REGION Network 3: Avoidance
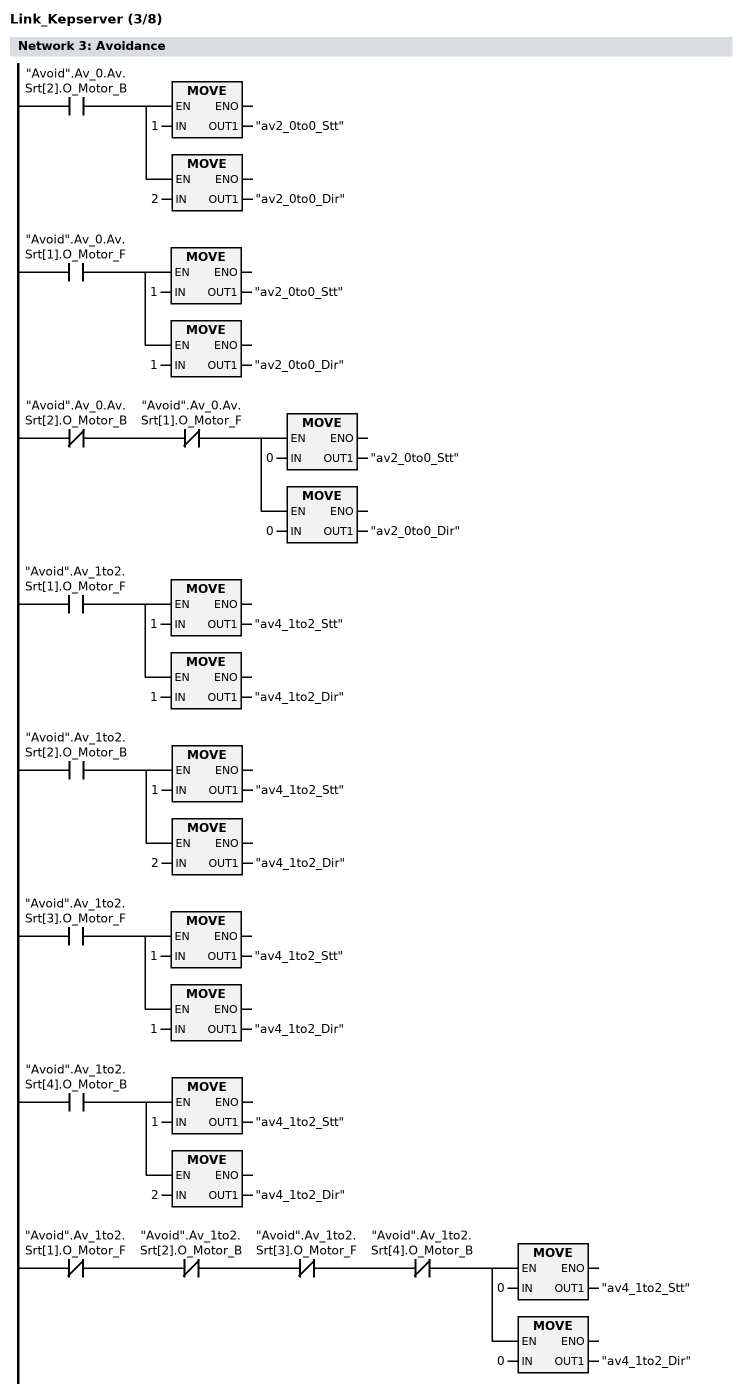
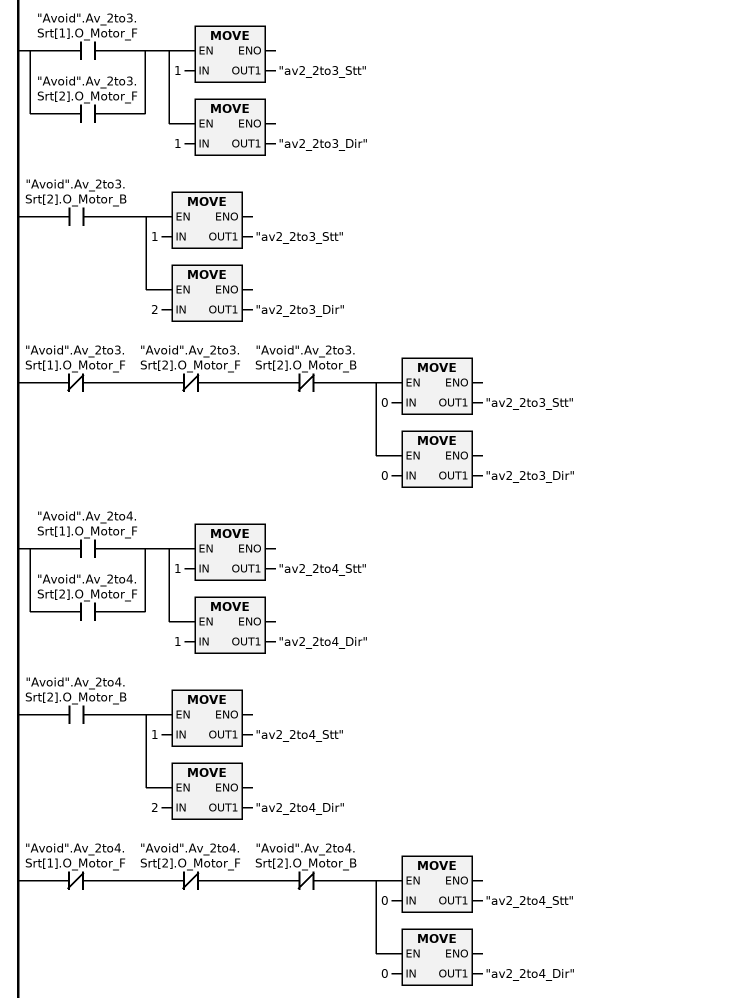
   RUNG wire#powerrail
      Contact( "Avoid".Av_0.Av.Srt[2].O_Motor_B )
      wire#w1
      Move(in := 1, out1 => "av2_0to0_Stt")
   END_RUNG
   RUNG wire#w1
      Move(in := 2, out1 => "av2_0to0_Dir")
   END_RUNG
   RUNG wire#powerrail
      Contact( "Avoid".Av_0.Av.Srt[1].O_Motor_F )
      wire#w2
      Move(in := 1, out1 => "av2_0to0_Stt")
   END_RUNG
   RUNG wire#w2
      Move(in := 1, out1 => "av2_0to0_Dir")
   END_RUNG
   RUNG wire#powerrail
      I_Contact( "Avoid".Av_0.Av.Srt[2].O_Motor_B )
      I_Contact( "Avoid".Av_0.Av.Srt[1].O_Motor_F )
      wire#w3
      Move(in := 0, out1 => "av2_0to0_Stt")
   END_RUNG
   RUNG wire#w3
      Move(in := 0, out1 => "av2_0to0_Dir")
   END_RUNG
   RUNG wire#powerrail
      Contact( "Avoid".Av_1to2.Srt[1].O_Motor_F )
      wire#w4
      Move(in := 1, out1 => "av4_1to2_Stt")
   END_RUNG
   RUNG wire#w4
      Move(in := 1, out1 => "av4_1to2_Dir")
   END_RUNG
   RUNG wire#powerrail
      Contact( "Avoid".Av_1to2.Srt[2].O_Motor_B )
      wire#w5
      Move(in := 1, out1 => "av4_1to2_Stt")
   END_RUNG
   RUNG wire#w5
      Move(in := 2, out1 => "av4_1to2_Dir")
   END_RUNG
   RUNG wire#powerrail
      Contact( "Avoid".Av_1to2.Srt[3].O_Motor_F )
      wire#w6
      Move(in := 1, out1 => "av4_1to2_Stt")
   END_RUNG
   RUNG wire#w6
      Move(in := 1, out1 => "av4_1to2_Dir")
   END_RUNG
   RUNG wire#powerrail
      Contact( "Avoid".Av_1to2.Srt[4].O_Motor_B )
      wire#w7
      Move(in := 1, out1 => "av4_1to2_Stt")
   END_RUNG
   RUNG wire#w7
      Move(in := 2, out1 => "av4_1to2_Dir")
   END_RUNG
   RUNG wire#powerrail
      I_Contact( "Avoid".Av_1to2.Srt[1].O_Motor_F )
      I_Contact( "Avoid".Av_1to2.Srt[2].O_Motor_B )
      I_Contact( "Avoid".Av_1to2.Srt[3].O_Motor_F )
      I_Contact( "Avoid".Av_1to2.Srt[4].O_Motor_B )
      wire#w8
      Move(in := 0, out1 => "av4_1to2_Stt")
   END_RUNG
   RUNG wire#w8
      Move(in := 0, out1 => "av4_1to2_Dir")
   END_RUNG
   RUNG wire#powerrail
      Contact( "Avoid".Av_2to3.Srt[1].O_Motor_F )
      wire#w9
      Move(in := 1, out1 => "av2_2to3_Stt")
   END_RUNG
   RUNG wire#powerrail
      Contact( "Avoid".Av_2to3.Srt[2].O_Motor_F )
   END_RUNG wire#w9
   RUNG wire#w9
      Move(in := 1, out1 => "av2_2to3_Dir")
   END_RUNG
   RUNG wire#powerrail
      Contact( "Avoid".Av_2to3.Srt[2].O_Motor_B )
      wire#w10
      Move(in := 1, out1 => "av2_2to3_Stt")
   END_RUNG
   RUNG wire#w10
      Move(in := 2, out1 => "av2_2to3_Dir")
   END_RUNG
   RUNG wire#powerrail
      I_Contact( "Avoid".Av_2to3.Srt[1].O_Motor_F )
      I_Contact( "Avoid".Av_2to3.Srt[2].O_Motor_F )
      I_Contact( "Avoid".Av_2to3.Srt[2].O_Motor_B )
      wire#w11
      Move(in := 0, out1 => "av2_2to3_Stt")
   END_RUNG
   RUNG wire#w11
      Move(in := 0, out1 => "av2_2to3_Dir")
   END_RUNG
   RUNG wire#powerrail
      Contact( "Avoid".Av_2to4.Srt[1].O_Motor_F )
      wire#w12
      Move(in := 1, out1 => "av2_2to4_Stt")
   END_RUNG
   RUNG wire#powerrail
      Contact( "Avoid".Av_2to4.Srt[2].O_Motor_F )
   END_RUNG wire#w12
   RUNG wire#w12
      Move(in := 1, out1 => "av2_2to4_Dir")
   END_RUNG
   RUNG wire#powerrail
      Contact( "Avoid".Av_2to4.Srt[2].O_Motor_B )
      wire#w13
      Move(in := 1, out1 => "av2_2to4_Stt")
   END_RUNG
   RUNG wire#w13
      Move(in := 2, out1 => "av2_2to4_Dir")
   END_RUNG
   RUNG wire#powerrail
      I_Contact( "Avoid".Av_2to4.Srt[1].O_Motor_F )
      I_Contact( "Avoid".Av_2to4.Srt[2].O_Motor_F )
      I_Contact( "Avoid".Av_2to4.Srt[2].O_Motor_B )
      wire#w14
      Move(in := 0, out1 => "av2_2to4_Stt")
   END_RUNG
   RUNG wire#w14
      Move(in := 0, out1 => "av2_2to4_Dir")
   END_RUNG
   // the same network as SCL:
   IF "Avoid".Av_0.Av.Srt[2].O_Motor_B THEN
       "av2_0to0_Stt" := 1;
       "av2_0to0_Dir" := 2;
   END_IF;
   IF "Avoid".Av_0.Av.Srt[1].O_Motor_F THEN
       "av2_0to0_Stt" := 1;
       "av2_0to0_Dir" := 1;
   END_IF;
   IF NOT "Avoid".Av_0.Av.Srt[2].O_Motor_B AND NOT "Avoid".Av_0.Av.Srt[1].O_Motor_F THEN
       "av2_0to0_Stt" := 0;
       "av2_0to0_Dir" := 0;
   END_IF;
   IF "Avoid".Av_1to2.Srt[1].O_Motor_F THEN
       "av4_1to2_Stt" := 1;
       "av4_1to2_Dir" := 1;
   END_IF;
   IF "Avoid".Av_1to2.Srt[2].O_Motor_B THEN
       "av4_1to2_Stt" := 1;
       "av4_1to2_Dir" := 2;
   END_IF;
   IF "Avoid".Av_1to2.Srt[3].O_Motor_F THEN
       "av4_1to2_Stt" := 1;
       "av4_1to2_Dir" := 1;
   END_IF;
   IF "Avoid".Av_1to2.Srt[4].O_Motor_B THEN
       "av4_1to2_Stt" := 1;
       "av4_1to2_Dir" := 2;
   END_IF;
   IF NOT "Avoid".Av_1to2.Srt[1].O_Motor_F AND NOT "Avoid".Av_1to2.Srt[2].O_Motor_B AND NOT "Avoid".Av_1to2.Srt[3].O_Motor_F AND NOT "Avoid".Av_1to2.Srt[4].O_Motor_B THEN
       "av4_1to2_Stt" := 0;
       "av4_1to2_Dir" := 0;
   END_IF;
   IF "Avoid".Av_2to3.Srt[1].O_Motor_F OR "Avoid".Av_2to3.Srt[2].O_Motor_F THEN
       "av2_2to3_Stt" := 1;
       "av2_2to3_Dir" := 1;
   END_IF;
   IF "Avoid".Av_2to3.Srt[2].O_Motor_B THEN
       "av2_2to3_Stt" := 1;
       "av2_2to3_Dir" := 2;
   END_IF;
   IF NOT "Avoid".Av_2to3.Srt[1].O_Motor_F AND NOT "Avoid".Av_2to3.Srt[2].O_Motor_F AND NOT "Avoid".Av_2to3.Srt[2].O_Motor_B THEN
       "av2_2to3_Stt" := 0;
       "av2_2to3_Dir" := 0;
   END_IF;
   IF "Avoid".Av_2to4.Srt[1].O_Motor_F OR "Avoid".Av_2to4.Srt[2].O_Motor_F THEN
       "av2_2to4_Stt" := 1;
       "av2_2to4_Dir" := 1;
   END_IF;
   IF "Avoid".Av_2to4.Srt[2].O_Motor_B THEN
       "av2_2to4_Stt" := 1;
       "av2_2to4_Dir" := 2;
   END_IF;
   IF NOT "Avoid".Av_2to4.Srt[1].O_Motor_F AND NOT "Avoid".Av_2to4.Srt[2].O_Motor_F AND NOT "Avoid".Av_2to4.Srt[2].O_Motor_B THEN
       "av2_2to4_Stt" := 0;
       "av2_2to4_Dir" := 0;
   END_IF;
END_REGION

REGION Network 4: Updown
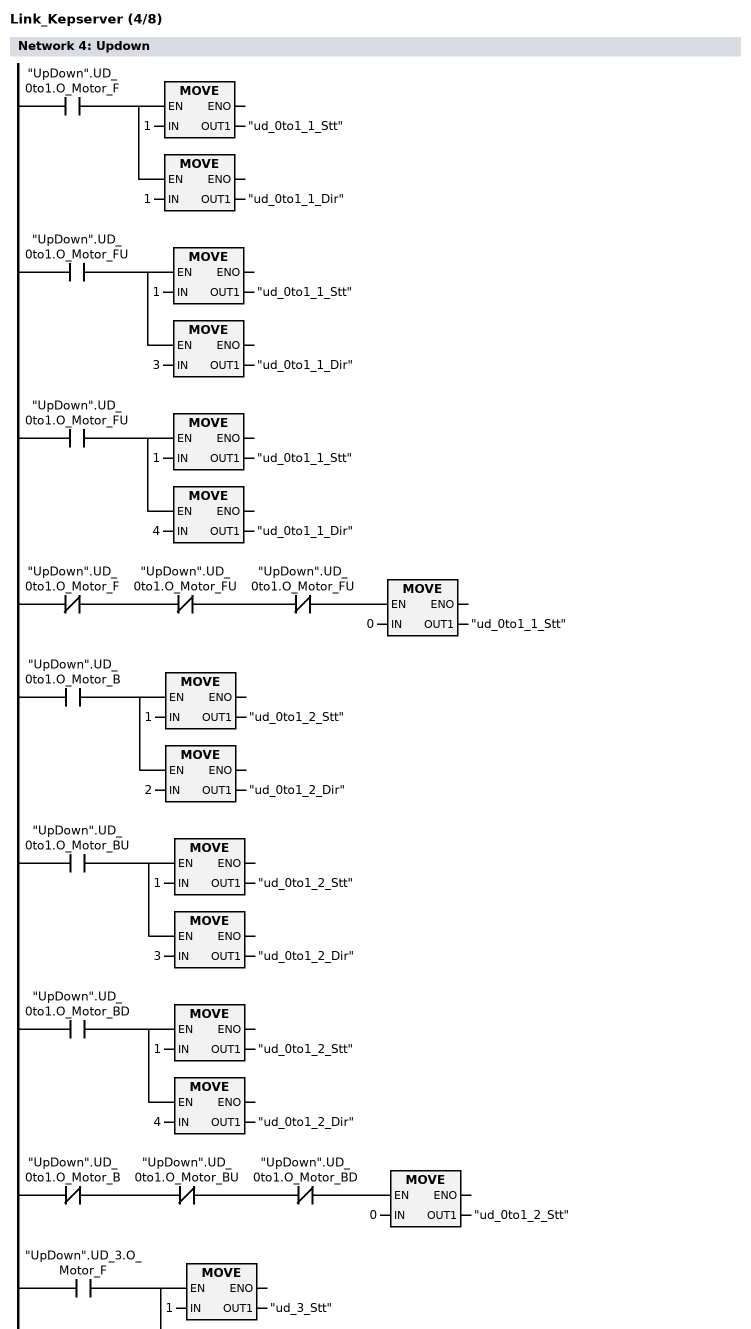
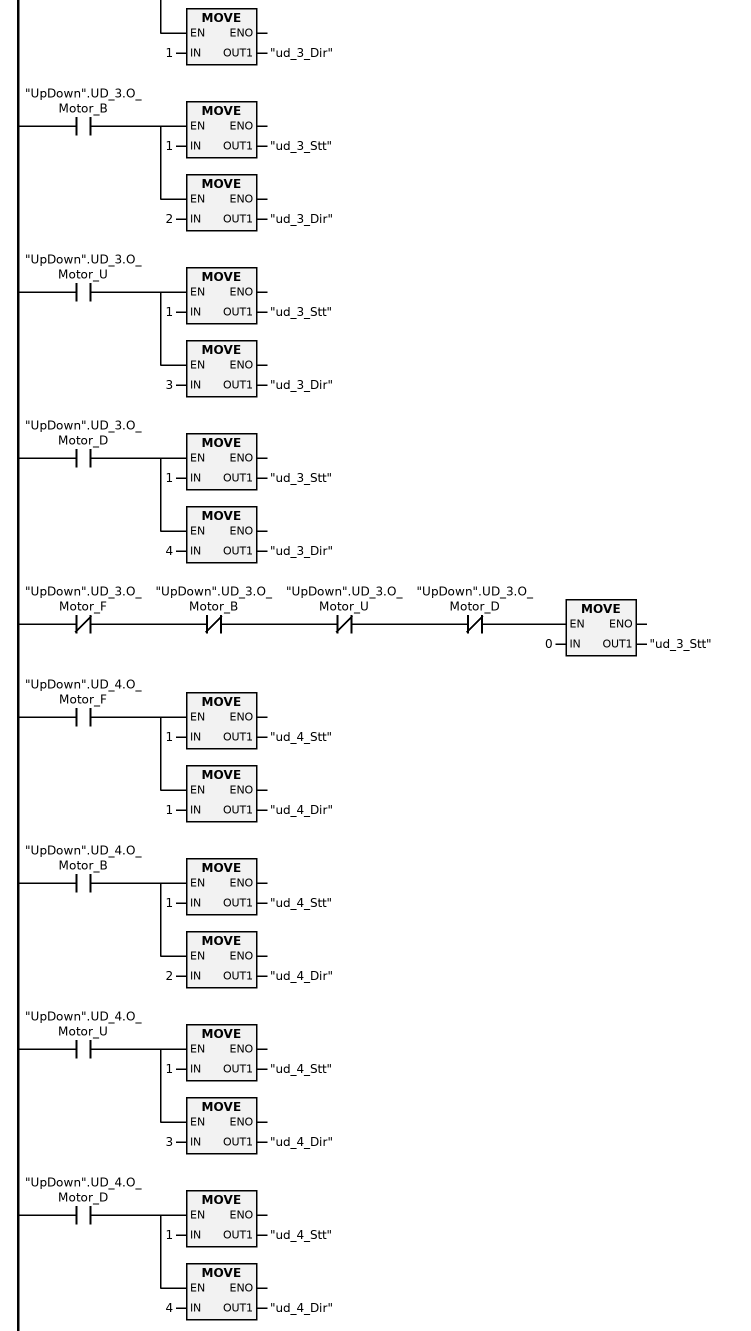
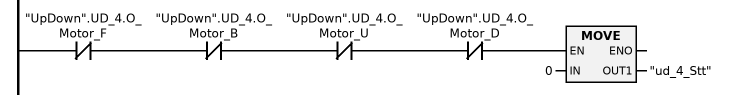
   RUNG wire#powerrail
      Contact( "UpDown".UD_0to1.O_Motor_F )
      wire#w1
      Move(in := 1, out1 => "ud_0to1_1_Stt")
   END_RUNG
   RUNG wire#w1
      Move(in := 1, out1 => "ud_0to1_1_Dir")
   END_RUNG
   RUNG wire#powerrail
      Contact( "UpDown".UD_0to1.O_Motor_FU )
      wire#w2
      Move(in := 1, out1 => "ud_0to1_1_Stt")
   END_RUNG
   RUNG wire#w2
      Move(in := 3, out1 => "ud_0to1_1_Dir")
   END_RUNG
   RUNG wire#powerrail
      Contact( "UpDown".UD_0to1.O_Motor_FU )
      wire#w3
      Move(in := 1, out1 => "ud_0to1_1_Stt")
   END_RUNG
   RUNG wire#w3
      Move(in := 4, out1 => "ud_0to1_1_Dir")
   END_RUNG
   RUNG wire#powerrail
      I_Contact( "UpDown".UD_0to1.O_Motor_F )
      I_Contact( "UpDown".UD_0to1.O_Motor_FU )
      I_Contact( "UpDown".UD_0to1.O_Motor_FU )
      Move(in := 0, out1 => "ud_0to1_1_Stt")
   END_RUNG
   RUNG wire#powerrail
      Contact( "UpDown".UD_0to1.O_Motor_B )
      wire#w4
      Move(in := 1, out1 => "ud_0to1_2_Stt")
   END_RUNG
   RUNG wire#w4
      Move(in := 2, out1 => "ud_0to1_2_Dir")
   END_RUNG
   RUNG wire#powerrail
      Contact( "UpDown".UD_0to1.O_Motor_BU )
      wire#w5
      Move(in := 1, out1 => "ud_0to1_2_Stt")
   END_RUNG
   RUNG wire#w5
      Move(in := 3, out1 => "ud_0to1_2_Dir")
   END_RUNG
   RUNG wire#powerrail
      Contact( "UpDown".UD_0to1.O_Motor_BD )
      wire#w6
      Move(in := 1, out1 => "ud_0to1_2_Stt")
   END_RUNG
   RUNG wire#w6
      Move(in := 4, out1 => "ud_0to1_2_Dir")
   END_RUNG
   RUNG wire#powerrail
      I_Contact( "UpDown".UD_0to1.O_Motor_B )
      I_Contact( "UpDown".UD_0to1.O_Motor_BU )
      I_Contact( "UpDown".UD_0to1.O_Motor_BD )
      Move(in := 0, out1 => "ud_0to1_2_Stt")
   END_RUNG
   RUNG wire#powerrail
      Contact( "UpDown".UD_3.O_Motor_F )
      wire#w7
      Move(in := 1, out1 => "ud_3_Stt")
   END_RUNG
   RUNG wire#w7
      Move(in := 1, out1 => "ud_3_Dir")
   END_RUNG
   RUNG wire#powerrail
      Contact( "UpDown".UD_3.O_Motor_B )
      wire#w8
      Move(in := 1, out1 => "ud_3_Stt")
   END_RUNG
   RUNG wire#w8
      Move(in := 2, out1 => "ud_3_Dir")
   END_RUNG
   RUNG wire#powerrail
      Contact( "UpDown".UD_3.O_Motor_U )
      wire#w9
      Move(in := 1, out1 => "ud_3_Stt")
   END_RUNG
   RUNG wire#w9
      Move(in := 3, out1 => "ud_3_Dir")
   END_RUNG
   RUNG wire#powerrail
      Contact( "UpDown".UD_3.O_Motor_D )
      wire#w10
      Move(in := 1, out1 => "ud_3_Stt")
   END_RUNG
   RUNG wire#w10
      Move(in := 4, out1 => "ud_3_Dir")
   END_RUNG
   RUNG wire#powerrail
      I_Contact( "UpDown".UD_3.O_Motor_F )
      I_Contact( "UpDown".UD_3.O_Motor_B )
      I_Contact( "UpDown".UD_3.O_Motor_U )
      I_Contact( "UpDown".UD_3.O_Motor_D )
      Move(in := 0, out1 => "ud_3_Stt")
   END_RUNG
   RUNG wire#powerrail
      Contact( "UpDown".UD_4.O_Motor_F )
      wire#w11
      Move(in := 1, out1 => "ud_4_Stt")
   END_RUNG
   RUNG wire#w11
      Move(in := 1, out1 => "ud_4_Dir")
   END_RUNG
   RUNG wire#powerrail
      Contact( "UpDown".UD_4.O_Motor_B )
      wire#w12
      Move(in := 1, out1 => "ud_4_Stt")
   END_RUNG
   RUNG wire#w12
      Move(in := 2, out1 => "ud_4_Dir")
   END_RUNG
   RUNG wire#powerrail
      Contact( "UpDown".UD_4.O_Motor_U )
      wire#w13
      Move(in := 1, out1 => "ud_4_Stt")
   END_RUNG
   RUNG wire#w13
      Move(in := 3, out1 => "ud_4_Dir")
   END_RUNG
   RUNG wire#powerrail
      Contact( "UpDown".UD_4.O_Motor_D )
      wire#w14
      Move(in := 1, out1 => "ud_4_Stt")
   END_RUNG
   RUNG wire#w14
      Move(in := 4, out1 => "ud_4_Dir")
   END_RUNG
   RUNG wire#powerrail
      I_Contact( "UpDown".UD_4.O_Motor_F )
      I_Contact( "UpDown".UD_4.O_Motor_B )
      I_Contact( "UpDown".UD_4.O_Motor_U )
      I_Contact( "UpDown".UD_4.O_Motor_D )
      Move(in := 0, out1 => "ud_4_Stt")
   END_RUNG
   // the same network as SCL:
   IF "UpDown".UD_0to1.O_Motor_F THEN
       "ud_0to1_1_Stt" := 1;
       "ud_0to1_1_Dir" := 1;
   END_IF;
   IF "UpDown".UD_0to1.O_Motor_FU THEN
       "ud_0to1_1_Stt" := 1;
       "ud_0to1_1_Dir" := 3;
       "ud_0to1_1_Stt" := 1;
       "ud_0to1_1_Dir" := 4;
   END_IF;
   IF NOT "UpDown".UD_0to1.O_Motor_F AND NOT "UpDown".UD_0to1.O_Motor_FU AND NOT "UpDown".UD_0to1.O_Motor_FU THEN
       "ud_0to1_1_Stt" := 0;
   END_IF;
   IF "UpDown".UD_0to1.O_Motor_B THEN
       "ud_0to1_2_Stt" := 1;
       "ud_0to1_2_Dir" := 2;
   END_IF;
   IF "UpDown".UD_0to1.O_Motor_BU THEN
       "ud_0to1_2_Stt" := 1;
       "ud_0to1_2_Dir" := 3;
   END_IF;
   IF "UpDown".UD_0to1.O_Motor_BD THEN
       "ud_0to1_2_Stt" := 1;
       "ud_0to1_2_Dir" := 4;
   END_IF;
   IF NOT "UpDown".UD_0to1.O_Motor_B AND NOT "UpDown".UD_0to1.O_Motor_BU AND NOT "UpDown".UD_0to1.O_Motor_BD THEN
       "ud_0to1_2_Stt" := 0;
   END_IF;
   IF "UpDown".UD_3.O_Motor_F THEN
       "ud_3_Stt" := 1;
       "ud_3_Dir" := 1;
   END_IF;
   IF "UpDown".UD_3.O_Motor_B THEN
       "ud_3_Stt" := 1;
       "ud_3_Dir" := 2;
   END_IF;
   IF "UpDown".UD_3.O_Motor_U THEN
       "ud_3_Stt" := 1;
       "ud_3_Dir" := 3;
   END_IF;
   IF "UpDown".UD_3.O_Motor_D THEN
       "ud_3_Stt" := 1;
       "ud_3_Dir" := 4;
   END_IF;
   IF NOT "UpDown".UD_3.O_Motor_F AND NOT "UpDown".UD_3.O_Motor_B AND NOT "UpDown".UD_3.O_Motor_U AND NOT "UpDown".UD_3.O_Motor_D THEN
       "ud_3_Stt" := 0;
   END_IF;
   IF "UpDown".UD_4.O_Motor_F THEN
       "ud_4_Stt" := 1;
       "ud_4_Dir" := 1;
   END_IF;
   IF "UpDown".UD_4.O_Motor_B THEN
       "ud_4_Stt" := 1;
       "ud_4_Dir" := 2;
   END_IF;
   IF "UpDown".UD_4.O_Motor_U THEN
       "ud_4_Stt" := 1;
       "ud_4_Dir" := 3;
   END_IF;
   IF "UpDown".UD_4.O_Motor_D THEN
       "ud_4_Stt" := 1;
       "ud_4_Dir" := 4;
   END_IF;
   IF NOT "UpDown".UD_4.O_Motor_F AND NOT "UpDown".UD_4.O_Motor_B AND NOT "UpDown".UD_4.O_Motor_U AND NOT "UpDown".UD_4.O_Motor_D THEN
       "ud_4_Stt" := 0;
   END_IF;
END_REGION

REGION Network 5: LS_Avoidance
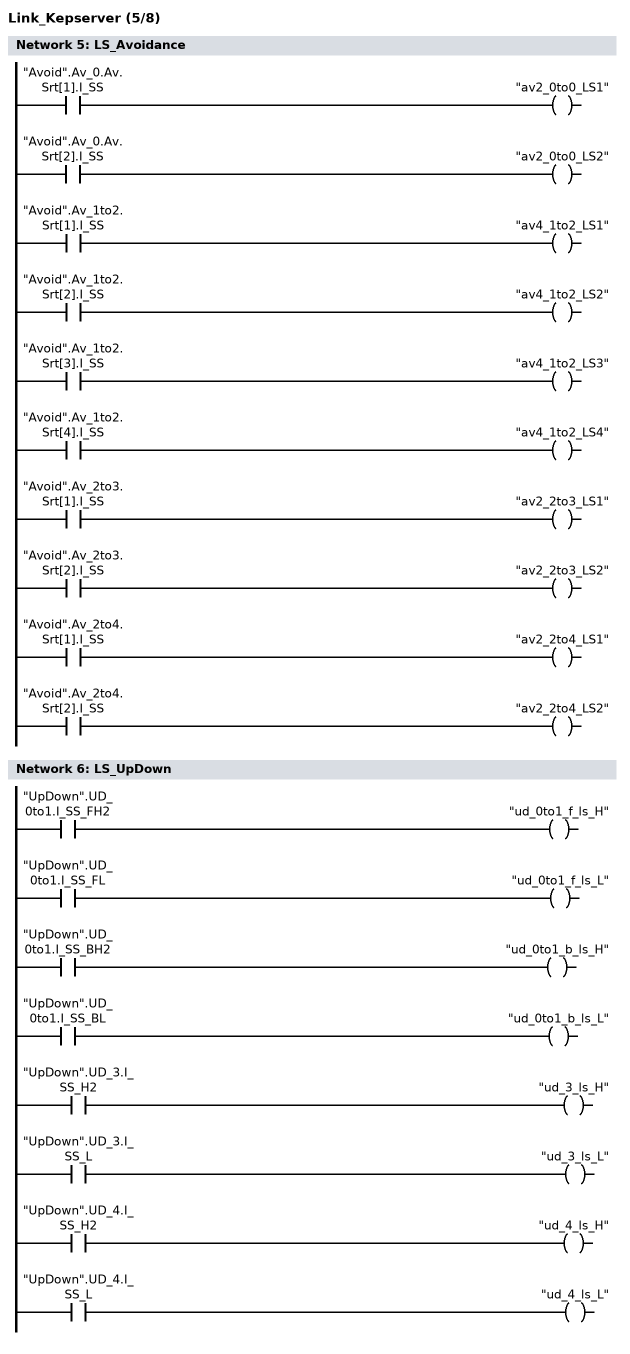
   RUNG wire#powerrail
      Contact( "Avoid".Av_0.Av.Srt[1].I_SS )
      Coil( "av2_0to0_LS1" )
   END_RUNG
   RUNG wire#powerrail
      Contact( "Avoid".Av_0.Av.Srt[2].I_SS )
      Coil( "av2_0to0_LS2" )
   END_RUNG
   RUNG wire#powerrail
      Contact( "Avoid".Av_1to2.Srt[1].I_SS )
      Coil( "av4_1to2_LS1" )
   END_RUNG
   RUNG wire#powerrail
      Contact( "Avoid".Av_1to2.Srt[2].I_SS )
      Coil( "av4_1to2_LS2" )
   END_RUNG
   RUNG wire#powerrail
      Contact( "Avoid".Av_1to2.Srt[3].I_SS )
      Coil( "av4_1to2_LS3" )
   END_RUNG
   RUNG wire#powerrail
      Contact( "Avoid".Av_1to2.Srt[4].I_SS )
      Coil( "av4_1to2_LS4" )
   END_RUNG
   RUNG wire#powerrail
      Contact( "Avoid".Av_2to3.Srt[1].I_SS )
      Coil( "av2_2to3_LS1" )
   END_RUNG
   RUNG wire#powerrail
      Contact( "Avoid".Av_2to3.Srt[2].I_SS )
      Coil( "av2_2to3_LS2" )
   END_RUNG
   RUNG wire#powerrail
      Contact( "Avoid".Av_2to4.Srt[1].I_SS )
      Coil( "av2_2to4_LS1" )
   END_RUNG
   RUNG wire#powerrail
      Contact( "Avoid".Av_2to4.Srt[2].I_SS )
      Coil( "av2_2to4_LS2" )
   END_RUNG
   // the same network as SCL:
   "av2_0to0_LS1" := "Avoid".Av_0.Av.Srt[1].I_SS;
   "av2_0to0_LS2" := "Avoid".Av_0.Av.Srt[2].I_SS;
   "av4_1to2_LS1" := "Avoid".Av_1to2.Srt[1].I_SS;
   "av4_1to2_LS2" := "Avoid".Av_1to2.Srt[2].I_SS;
   "av4_1to2_LS3" := "Avoid".Av_1to2.Srt[3].I_SS;
   "av4_1to2_LS4" := "Avoid".Av_1to2.Srt[4].I_SS;
   "av2_2to3_LS1" := "Avoid".Av_2to3.Srt[1].I_SS;
   "av2_2to3_LS2" := "Avoid".Av_2to3.Srt[2].I_SS;
   "av2_2to4_LS1" := "Avoid".Av_2to4.Srt[1].I_SS;
   "av2_2to4_LS2" := "Avoid".Av_2to4.Srt[2].I_SS;
END_REGION

REGION Network 6: LS_UpDown
   RUNG wire#powerrail
      Contact( "UpDown".UD_0to1.I_SS_FH2 )
      Coil( "ud_0to1_f_ls_H" )
   END_RUNG
   RUNG wire#powerrail
      Contact( "UpDown".UD_0to1.I_SS_FL )
      Coil( "ud_0to1_f_ls_L" )
   END_RUNG
   RUNG wire#powerrail
      Contact( "UpDown".UD_0to1.I_SS_BH2 )
      Coil( "ud_0to1_b_ls_H" )
   END_RUNG
   RUNG wire#powerrail
      Contact( "UpDown".UD_0to1.I_SS_BL )
      Coil( "ud_0to1_b_ls_L" )
   END_RUNG
   RUNG wire#powerrail
      Contact( "UpDown".UD_3.I_SS_H2 )
      Coil( "ud_3_ls_H" )
   END_RUNG
   RUNG wire#powerrail
      Contact( "UpDown".UD_3.I_SS_L )
      Coil( "ud_3_ls_L" )
   END_RUNG
   RUNG wire#powerrail
      Contact( "UpDown".UD_4.I_SS_H2 )
      Coil( "ud_4_ls_H" )
   END_RUNG
   RUNG wire#powerrail
      Contact( "UpDown".UD_4.I_SS_L )
      Coil( "ud_4_ls_L" )
   END_RUNG
   // the same network as SCL:
   "ud_0to1_f_ls_H" := "UpDown".UD_0to1.I_SS_FH2;
   "ud_0to1_f_ls_L" := "UpDown".UD_0to1.I_SS_FL;
   "ud_0to1_b_ls_H" := "UpDown".UD_0to1.I_SS_BH2;
   "ud_0to1_b_ls_L" := "UpDown".UD_0to1.I_SS_BL;
   "ud_3_ls_H" := "UpDown".UD_3.I_SS_H2;
   "ud_3_ls_L" := "UpDown".UD_3.I_SS_L;
   "ud_4_ls_H" := "UpDown".UD_4.I_SS_H2;
   "ud_4_ls_L" := "UpDown".UD_4.I_SS_L;
END_REGION

REGION Network 7: Boxes _ cnv1d
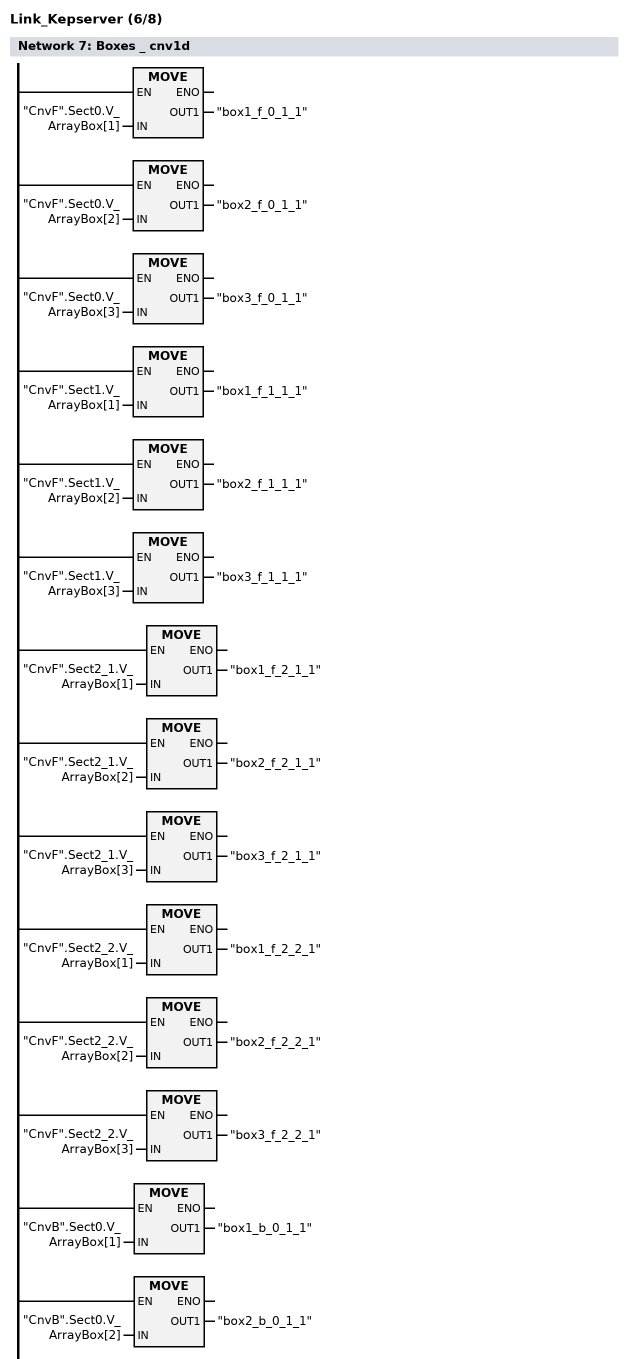
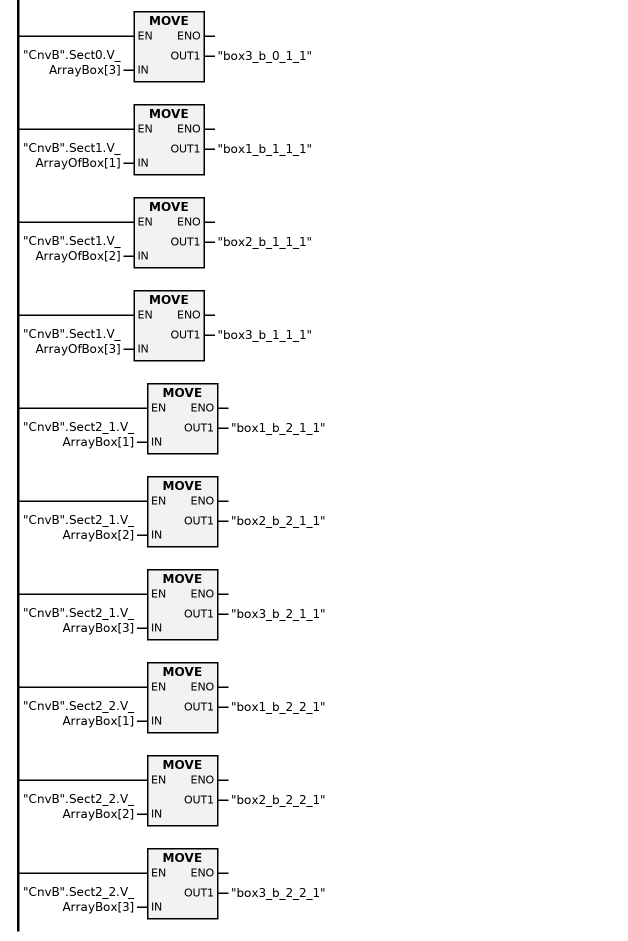
   RUNG wire#powerrail
      Move(in := "CnvF".Sect0.V_ArrayBox[1], out1 => "box1_f_0_1_1")
   END_RUNG
   RUNG wire#powerrail
      Move(in := "CnvF".Sect0.V_ArrayBox[2], out1 => "box2_f_0_1_1")
   END_RUNG
   RUNG wire#powerrail
      Move(in := "CnvF".Sect0.V_ArrayBox[3], out1 => "box3_f_0_1_1")
   END_RUNG
   RUNG wire#powerrail
      Move(in := "CnvF".Sect1.V_ArrayBox[1], out1 => "box1_f_1_1_1")
   END_RUNG
   RUNG wire#powerrail
      Move(in := "CnvF".Sect1.V_ArrayBox[2], out1 => "box2_f_1_1_1")
   END_RUNG
   RUNG wire#powerrail
      Move(in := "CnvF".Sect1.V_ArrayBox[3], out1 => "box3_f_1_1_1")
   END_RUNG
   RUNG wire#powerrail
      Move(in := "CnvF".Sect2_1.V_ArrayBox[1], out1 => "box1_f_2_1_1")
   END_RUNG
   RUNG wire#powerrail
      Move(in := "CnvF".Sect2_1.V_ArrayBox[2], out1 => "box2_f_2_1_1")
   END_RUNG
   RUNG wire#powerrail
      Move(in := "CnvF".Sect2_1.V_ArrayBox[3], out1 => "box3_f_2_1_1")
   END_RUNG
   RUNG wire#powerrail
      Move(in := "CnvF".Sect2_2.V_ArrayBox[1], out1 => "box1_f_2_2_1")
   END_RUNG
   RUNG wire#powerrail
      Move(in := "CnvF".Sect2_2.V_ArrayBox[2], out1 => "box2_f_2_2_1")
   END_RUNG
   RUNG wire#powerrail
      Move(in := "CnvF".Sect2_2.V_ArrayBox[3], out1 => "box3_f_2_2_1")
   END_RUNG
   RUNG wire#powerrail
      Move(in := "CnvB".Sect0.V_ArrayBox[1], out1 => "box1_b_0_1_1")
   END_RUNG
   RUNG wire#powerrail
      Move(in := "CnvB".Sect0.V_ArrayBox[2], out1 => "box2_b_0_1_1")
   END_RUNG
   RUNG wire#powerrail
      Move(in := "CnvB".Sect0.V_ArrayBox[3], out1 => "box3_b_0_1_1")
   END_RUNG
   RUNG wire#powerrail
      Move(in := "CnvB".Sect1.V_ArrayOfBox[1], out1 => "box1_b_1_1_1")
   END_RUNG
   RUNG wire#powerrail
      Move(in := "CnvB".Sect1.V_ArrayOfBox[2], out1 => "box2_b_1_1_1")
   END_RUNG
   RUNG wire#powerrail
      Move(in := "CnvB".Sect1.V_ArrayOfBox[3], out1 => "box3_b_1_1_1")
   END_RUNG
   RUNG wire#powerrail
      Move(in := "CnvB".Sect2_1.V_ArrayBox[1], out1 => "box1_b_2_1_1")
   END_RUNG
   RUNG wire#powerrail
      Move(in := "CnvB".Sect2_1.V_ArrayBox[2], out1 => "box2_b_2_1_1")
   END_RUNG
   RUNG wire#powerrail
      Move(in := "CnvB".Sect2_1.V_ArrayBox[3], out1 => "box3_b_2_1_1")
   END_RUNG
   RUNG wire#powerrail
      Move(in := "CnvB".Sect2_2.V_ArrayBox[1], out1 => "box1_b_2_2_1")
   END_RUNG
   RUNG wire#powerrail
      Move(in := "CnvB".Sect2_2.V_ArrayBox[2], out1 => "box2_b_2_2_1")
   END_RUNG
   RUNG wire#powerrail
      Move(in := "CnvB".Sect2_2.V_ArrayBox[3], out1 => "box3_b_2_2_1")
   END_RUNG
   // the same network as SCL:
   "box1_f_0_1_1" := "CnvF".Sect0.V_ArrayBox[1];
   "box2_f_0_1_1" := "CnvF".Sect0.V_ArrayBox[2];
   "box3_f_0_1_1" := "CnvF".Sect0.V_ArrayBox[3];
   "box1_f_1_1_1" := "CnvF".Sect1.V_ArrayBox[1];
   "box2_f_1_1_1" := "CnvF".Sect1.V_ArrayBox[2];
   "box3_f_1_1_1" := "CnvF".Sect1.V_ArrayBox[3];
   "box1_f_2_1_1" := "CnvF".Sect2_1.V_ArrayBox[1];
   "box2_f_2_1_1" := "CnvF".Sect2_1.V_ArrayBox[2];
   "box3_f_2_1_1" := "CnvF".Sect2_1.V_ArrayBox[3];
   "box1_f_2_2_1" := "CnvF".Sect2_2.V_ArrayBox[1];
   "box2_f_2_2_1" := "CnvF".Sect2_2.V_ArrayBox[2];
   "box3_f_2_2_1" := "CnvF".Sect2_2.V_ArrayBox[3];
   "box1_b_0_1_1" := "CnvB".Sect0.V_ArrayBox[1];
   "box2_b_0_1_1" := "CnvB".Sect0.V_ArrayBox[2];
   "box3_b_0_1_1" := "CnvB".Sect0.V_ArrayBox[3];
   "box1_b_1_1_1" := "CnvB".Sect1.V_ArrayOfBox[1];
   "box2_b_1_1_1" := "CnvB".Sect1.V_ArrayOfBox[2];
   "box3_b_1_1_1" := "CnvB".Sect1.V_ArrayOfBox[3];
   "box1_b_2_1_1" := "CnvB".Sect2_1.V_ArrayBox[1];
   "box2_b_2_1_1" := "CnvB".Sect2_1.V_ArrayBox[2];
   "box3_b_2_1_1" := "CnvB".Sect2_1.V_ArrayBox[3];
   "box1_b_2_2_1" := "CnvB".Sect2_2.V_ArrayBox[1];
   "box2_b_2_2_1" := "CnvB".Sect2_2.V_ArrayBox[2];
   "box3_b_2_2_1" := "CnvB".Sect2_2.V_ArrayBox[3];
END_REGION

REGION Network 8: Boxes_Cnv2d
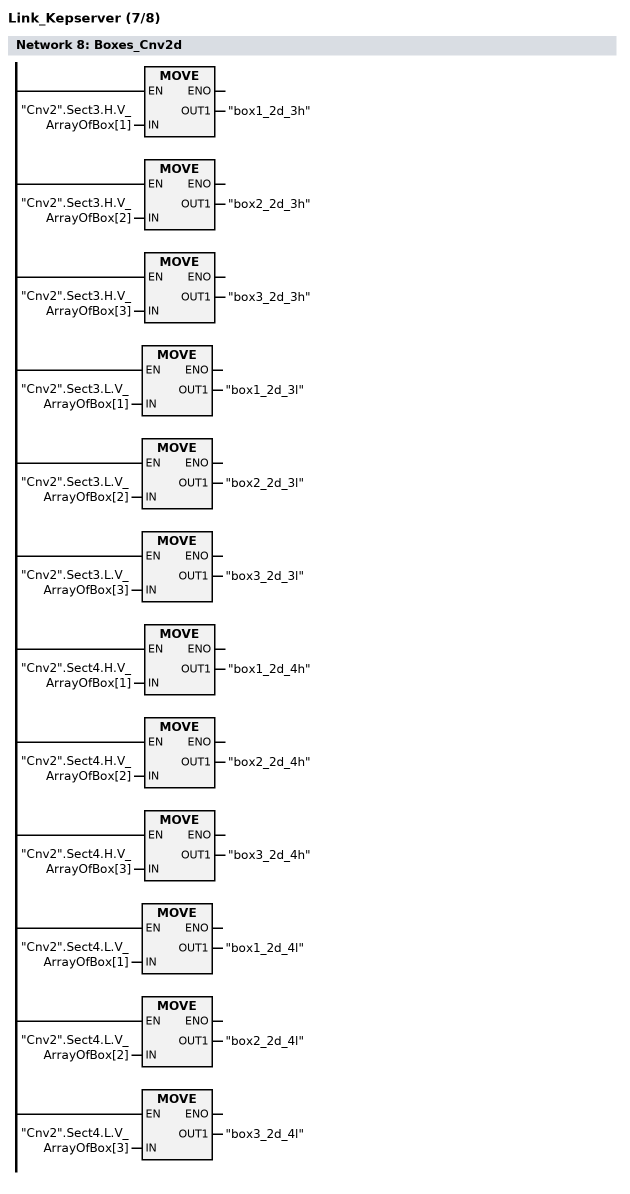
   RUNG wire#powerrail
      Move(in := "Cnv2".Sect3.H.V_ArrayOfBox[1], out1 => "box1_2d_3h")
   END_RUNG
   RUNG wire#powerrail
      Move(in := "Cnv2".Sect3.H.V_ArrayOfBox[2], out1 => "box2_2d_3h")
   END_RUNG
   RUNG wire#powerrail
      Move(in := "Cnv2".Sect3.H.V_ArrayOfBox[3], out1 => "box3_2d_3h")
   END_RUNG
   RUNG wire#powerrail
      Move(in := "Cnv2".Sect3.L.V_ArrayOfBox[1], out1 => "box1_2d_3l")
   END_RUNG
   RUNG wire#powerrail
      Move(in := "Cnv2".Sect3.L.V_ArrayOfBox[2], out1 => "box2_2d_3l")
   END_RUNG
   RUNG wire#powerrail
      Move(in := "Cnv2".Sect3.L.V_ArrayOfBox[3], out1 => "box3_2d_3l")
   END_RUNG
   RUNG wire#powerrail
      Move(in := "Cnv2".Sect4.H.V_ArrayOfBox[1], out1 => "box1_2d_4h")
   END_RUNG
   RUNG wire#powerrail
      Move(in := "Cnv2".Sect4.H.V_ArrayOfBox[2], out1 => "box2_2d_4h")
   END_RUNG
   RUNG wire#powerrail
      Move(in := "Cnv2".Sect4.H.V_ArrayOfBox[3], out1 => "box3_2d_4h")
   END_RUNG
   RUNG wire#powerrail
      Move(in := "Cnv2".Sect4.L.V_ArrayOfBox[1], out1 => "box1_2d_4l")
   END_RUNG
   RUNG wire#powerrail
      Move(in := "Cnv2".Sect4.L.V_ArrayOfBox[2], out1 => "box2_2d_4l")
   END_RUNG
   RUNG wire#powerrail
      Move(in := "Cnv2".Sect4.L.V_ArrayOfBox[3], out1 => "box3_2d_4l")
   END_RUNG
   // the same network as SCL:
   "box1_2d_3h" := "Cnv2".Sect3.H.V_ArrayOfBox[1];
   "box2_2d_3h" := "Cnv2".Sect3.H.V_ArrayOfBox[2];
   "box3_2d_3h" := "Cnv2".Sect3.H.V_ArrayOfBox[3];
   "box1_2d_3l" := "Cnv2".Sect3.L.V_ArrayOfBox[1];
   "box2_2d_3l" := "Cnv2".Sect3.L.V_ArrayOfBox[2];
   "box3_2d_3l" := "Cnv2".Sect3.L.V_ArrayOfBox[3];
   "box1_2d_4h" := "Cnv2".Sect4.H.V_ArrayOfBox[1];
   "box2_2d_4h" := "Cnv2".Sect4.H.V_ArrayOfBox[2];
   "box3_2d_4h" := "Cnv2".Sect4.H.V_ArrayOfBox[3];
   "box1_2d_4l" := "Cnv2".Sect4.L.V_ArrayOfBox[1];
   "box2_2d_4l" := "Cnv2".Sect4.L.V_ArrayOfBox[2];
   "box3_2d_4l" := "Cnv2".Sect4.L.V_ArrayOfBox[3];
END_REGION

REGION Network 9: Boxes_Av
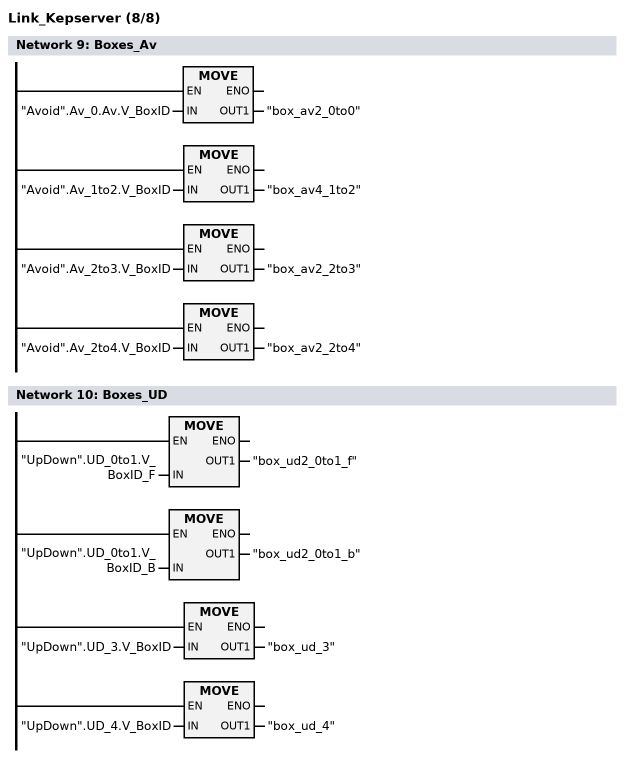
   RUNG wire#powerrail
      Move(in := "Avoid".Av_0.Av.V_BoxID, out1 => "box_av2_0to0")
   END_RUNG
   RUNG wire#powerrail
      Move(in := "Avoid".Av_1to2.V_BoxID, out1 => "box_av4_1to2")
   END_RUNG
   RUNG wire#powerrail
      Move(in := "Avoid".Av_2to3.V_BoxID, out1 => "box_av2_2to3")
   END_RUNG
   RUNG wire#powerrail
      Move(in := "Avoid".Av_2to4.V_BoxID, out1 => "box_av2_2to4")
   END_RUNG
   // the same network as SCL:
   "box_av2_0to0" := "Avoid".Av_0.Av.V_BoxID;
   "box_av4_1to2" := "Avoid".Av_1to2.V_BoxID;
   "box_av2_2to3" := "Avoid".Av_2to3.V_BoxID;
   "box_av2_2to4" := "Avoid".Av_2to4.V_BoxID;
END_REGION

REGION Network 10: Boxes_UD
   RUNG wire#powerrail
      Move(in := "UpDown".UD_0to1.V_BoxID_F, out1 => "box_ud2_0to1_f")
   END_RUNG
   RUNG wire#powerrail
      Move(in := "UpDown".UD_0to1.V_BoxID_B, out1 => "box_ud2_0to1_b")
   END_RUNG
   RUNG wire#powerrail
      Move(in := "UpDown".UD_3.V_BoxID, out1 => "box_ud_3")
   END_RUNG
   RUNG wire#powerrail
      Move(in := "UpDown".UD_4.V_BoxID, out1 => "box_ud_4")
   END_RUNG
   // the same network as SCL:
   "box_ud2_0to1_f" := "UpDown".UD_0to1.V_BoxID_F;
   "box_ud2_0to1_b" := "UpDown".UD_0to1.V_BoxID_B;
   "box_ud_3" := "UpDown".UD_3.V_BoxID;
   "box_ud_4" := "UpDown".UD_4.V_BoxID;
END_REGION
END_FUNCTION

FUNCTION "MHJ-PLC-Lab-Function-S71200" : Void   // FC9000, SCL
{ S7_Optimized_Access := 'TRUE' }
VERSION : 0.1
   VAR_TEMP
      rdTimeReturn : Int;
      outputTime : DTL;
      SyncVal : Byte;
      forVal : Int;
      forVal_2 : Int;
      Value : Byte;
   END_VAR
   VAR CONSTANT
      CompVal : Byte := 16#34;
      Value_01 : Byte := 16#11;
      Value_01_DW : DWord := 16#A165_D992;
      Value_02_DW : DWord := 16#58BE_4401;
   END_VAR
BEGIN

   #Value:=PEEK(area := 16#82,
        dbNumber := 0,
        byteOffset := 511);
   #Value := #Value + 1;

   POKE(area := 16#82,
        dbNumber := 0,
        byteOffset := 511,
        value := #Value);

   POKE(area:=16#81,
        dbNumber:=0,
        byteOffset:=1016,
        value:=#Value_01_DW);
   POKE(area := 16#81,
        dbNumber := 0,
        byteOffset := 1020,
        value := #Value_02_DW);

   POKE(area := 16#81,
        dbNumber := 0,
        byteOffset := 511,
        value := B#16#00);

   FOR #forVal := 0 TO 120 DO
       FOR #forVal_2:=0 TO 10 DO
           #rdTimeReturn:=RD_SYS_T(#outputTime);
           #rdTimeReturn := WR_SYS_T(#outputTime);
           #rdTimeReturn := RD_SYS_T(#outputTime);
           #rdTimeReturn := WR_SYS_T(#outputTime);
       END_FOR;
       #SyncVal:= PEEK(area := 16#81,
                      dbNumber := 0,
                      byteOffset := 511);
       IF #SyncVal = #CompVal THEN
          GOTO M_1;
       END_IF;
   END_FOR;
   RETURN;

   M_1:
   POKE(area := 16#81,
        dbNumber := 0,
        byteOffset := 511,
        value := B#16#0);
END_FUNCTION

ORGANIZATION_BLOCK "Main"   // OB1, LAD, ProgramCycle
TITLE = "Main Program Sweep (Cycle)"
{ S7_Optimized_Access := 'TRUE' }
VERSION : 0.1
   VAR_INPUT
      Initial_Call : Bool;   // Initial call of this OB
      Remanence : Bool;   // =True, if remanent data are available
   END_VAR
   VAR_TEMP   // added for the SCL form of the ladder/FBD networks
      _w1 : Bool;
      _w2 : Bool;
      _w3 : Bool;
      _w4 : Bool;
      _w5 : Bool;
      _w6 : Bool;
   END_VAR
BEGIN

REGION Network 1: Konnektierungsbaustein für PLC-Lab / Connect FtrIO
   // Im Netzwerk 1 wird der Konnektierungsbaustein für PLC-Lab aufgerufen.
   // Dieser Aufruf darf nicht entfernt werden!
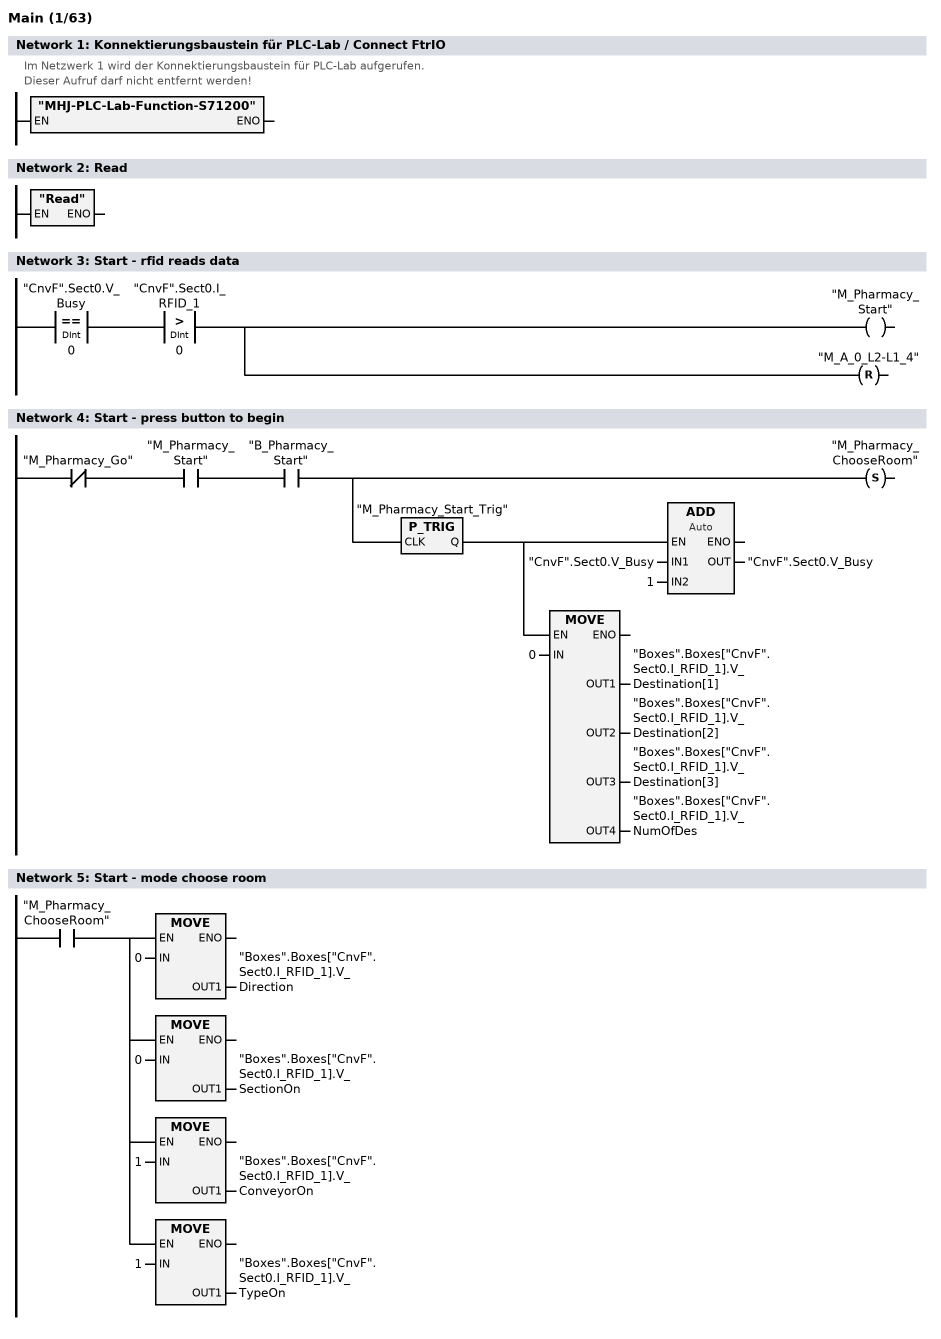
   RUNG wire#powerrail
      "MHJ-PLC-Lab-Function-S71200"()
   END_RUNG
   // the same network as SCL:
   "MHJ-PLC-Lab-Function-S71200"();
END_REGION

REGION Network 2: Read
   RUNG wire#powerrail
      "Read"()
   END_RUNG
   // the same network as SCL:
   "Read"();
END_REGION

REGION Network 3: Start - rfid reads data
   RUNG wire#powerrail
      { S7_Templates := "SrcType := DInt" } EQ_Contact(in1 := "CnvF".Sect0.V_Busy, in2 := 0)
      { S7_Templates := "SrcType := DInt" } GT_Contact(in1 := "CnvF".Sect0.I_RFID_1, in2 := 0)
      wire#w1
      Coil( "M_Pharmacy_Start" )
   END_RUNG
   RUNG wire#w1
      R_Coil( "M_A_0_L2-L1_4" )
   END_RUNG
   // the same network as SCL:
   "M_Pharmacy_Start" := ("CnvF".Sect0.V_Busy = 0) AND ("CnvF".Sect0.I_RFID_1 > 0);
   IF "M_Pharmacy_Start" THEN "M_A_0_L2-L1_4" := FALSE; END_IF;
END_REGION

REGION Network 4: Start - press button to begin
   RUNG wire#powerrail
      I_Contact( "M_Pharmacy_Go" )
      Contact( "M_Pharmacy_Start" )
      Contact( "B_Pharmacy_Start" )
      wire#w1
      S_Coil( "M_Pharmacy_ChooseRoom" )
   END_RUNG
   RUNG wire#w1
      P_Trig( "M_Pharmacy_Start_Trig" )
      wire#w2
      Add(in1 := "CnvF".Sect0.V_Busy, in2 := 1, out => "CnvF".Sect0.V_Busy)
   END_RUNG
   RUNG wire#w2
      Move(in := 0, out1 => "Boxes".Boxes["CnvF".Sect0.I_RFID_1].V_Destination[1], out2 => "Boxes".Boxes["CnvF".Sect0.I_RFID_1].V_Destination[2], out3 => "Boxes".Boxes["CnvF".Sect0.I_RFID_1].V_Destination[3], out4 => "Boxes".Boxes["CnvF".Sect0.I_RFID_1].V_NumOfDes)
   END_RUNG
   // the same network as SCL:
   #_w1 := NOT "M_Pharmacy_Go" AND "M_Pharmacy_Start" AND "B_Pharmacy_Start";
   IF #_w1 THEN "M_Pharmacy_ChooseRoom" := TRUE; END_IF;
   #_w2 := #_w1 AND NOT "M_Pharmacy_Start_Trig";   // rising edge
   "M_Pharmacy_Start_Trig" := #_w1;
   IF #_w2 THEN
       "CnvF".Sect0.V_Busy := "CnvF".Sect0.V_Busy + 1;
       "Boxes".Boxes["CnvF".Sect0.I_RFID_1].V_Destination[1] := 0;
       "Boxes".Boxes["CnvF".Sect0.I_RFID_1].V_Destination[2] := 0;
       "Boxes".Boxes["CnvF".Sect0.I_RFID_1].V_Destination[3] := 0;
       "Boxes".Boxes["CnvF".Sect0.I_RFID_1].V_NumOfDes := 0;
   END_IF;
END_REGION

REGION Network 5: Start - mode choose room
   RUNG wire#powerrail
      Contact( "M_Pharmacy_ChooseRoom" )
      wire#w1
      Move(in := 0, out1 => "Boxes".Boxes["CnvF".Sect0.I_RFID_1].V_Direction)
   END_RUNG
   RUNG wire#w1
      Move(in := 0, out1 => "Boxes".Boxes["CnvF".Sect0.I_RFID_1].V_SectionOn)
   END_RUNG
   RUNG wire#w1
      Move(in := 1, out1 => "Boxes".Boxes["CnvF".Sect0.I_RFID_1].V_ConveyorOn)
   END_RUNG
   RUNG wire#w1
      Move(in := 1, out1 => "Boxes".Boxes["CnvF".Sect0.I_RFID_1].V_TypeOn)
   END_RUNG
   // the same network as SCL:
   IF "M_Pharmacy_ChooseRoom" THEN
       "Boxes".Boxes["CnvF".Sect0.I_RFID_1].V_Direction := 0;
       "Boxes".Boxes["CnvF".Sect0.I_RFID_1].V_SectionOn := 0;
       "Boxes".Boxes["CnvF".Sect0.I_RFID_1].V_ConveyorOn := 1;
       "Boxes".Boxes["CnvF".Sect0.I_RFID_1].V_TypeOn := 1;
   END_IF;
END_REGION

REGION Network 6: Start - choose room
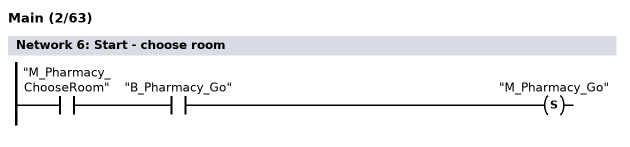
   RUNG wire#powerrail
      Contact( "M_Pharmacy_ChooseRoom" )
      Contact( "B_Pharmacy_Go" )
      S_Coil( "M_Pharmacy_Go" )
   END_RUNG
   // the same network as SCL:
   IF "M_Pharmacy_ChooseRoom" AND "B_Pharmacy_Go" THEN "M_Pharmacy_Go" := TRUE; END_IF;
END_REGION

REGION Network 7: Start - mode go
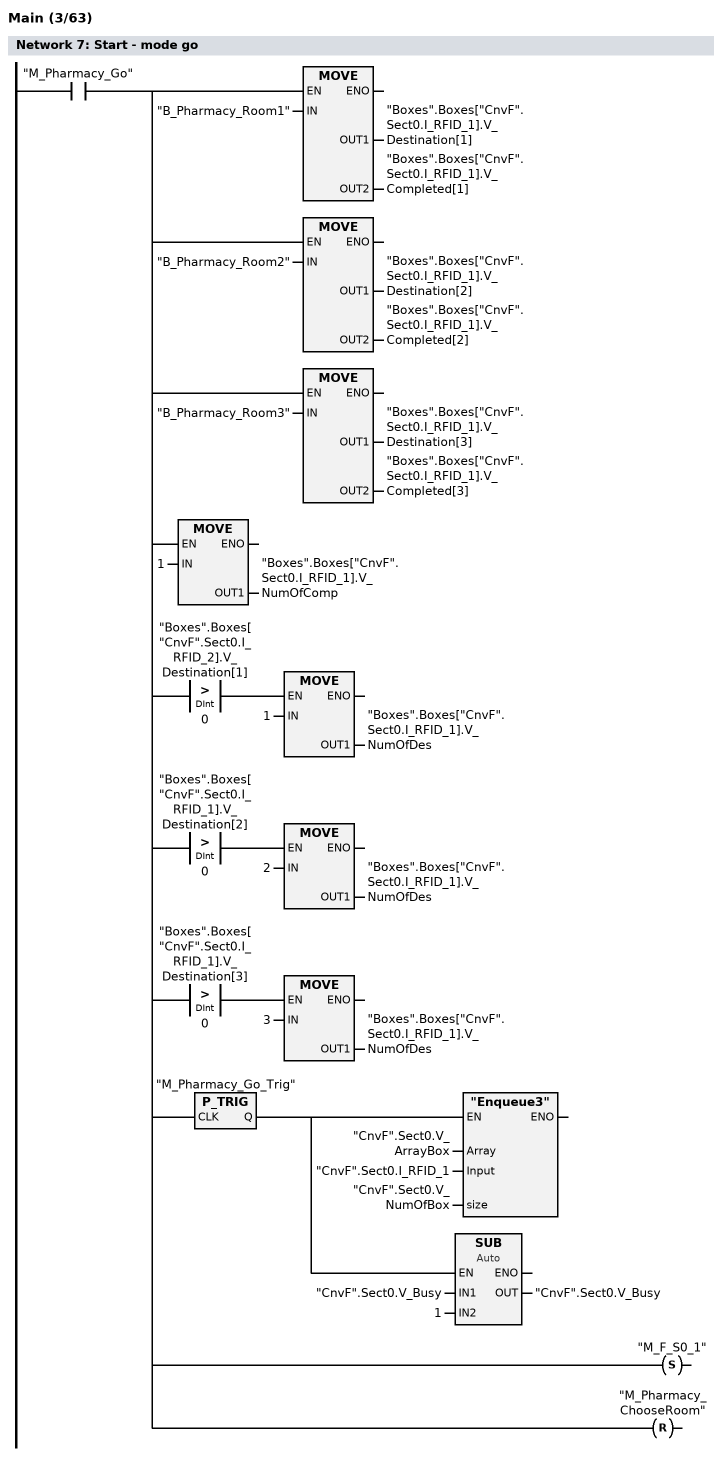
   RUNG wire#powerrail
      Contact( "M_Pharmacy_Go" )
      wire#w1
      Move(in := "B_Pharmacy_Room1", out1 => "Boxes".Boxes["CnvF".Sect0.I_RFID_1].V_Destination[1], out2 => "Boxes".Boxes["CnvF".Sect0.I_RFID_1].V_Completed[1])
   END_RUNG
   RUNG wire#w1
      Move(in := "B_Pharmacy_Room2", out1 => "Boxes".Boxes["CnvF".Sect0.I_RFID_1].V_Destination[2], out2 => "Boxes".Boxes["CnvF".Sect0.I_RFID_1].V_Completed[2])
   END_RUNG
   RUNG wire#w1
      Move(in := "B_Pharmacy_Room3", out1 => "Boxes".Boxes["CnvF".Sect0.I_RFID_1].V_Destination[3], out2 => "Boxes".Boxes["CnvF".Sect0.I_RFID_1].V_Completed[3])
   END_RUNG
   RUNG wire#w1
      Move(in := 1, out1 => "Boxes".Boxes["CnvF".Sect0.I_RFID_1].V_NumOfComp)
   END_RUNG
   RUNG wire#w1
      { S7_Templates := "SrcType := DInt" } GT_Contact(in1 := "Boxes".Boxes["CnvF".Sect0.I_RFID_2].V_Destination[1], in2 := 0)
      Move(in := 1, out1 => "Boxes".Boxes["CnvF".Sect0.I_RFID_1].V_NumOfDes)
   END_RUNG
   RUNG wire#w1
      { S7_Templates := "SrcType := DInt" } GT_Contact(in1 := "Boxes".Boxes["CnvF".Sect0.I_RFID_1].V_Destination[2], in2 := 0)
      Move(in := 2, out1 => "Boxes".Boxes["CnvF".Sect0.I_RFID_1].V_NumOfDes)
   END_RUNG
   RUNG wire#w1
      { S7_Templates := "SrcType := DInt" } GT_Contact(in1 := "Boxes".Boxes["CnvF".Sect0.I_RFID_1].V_Destination[3], in2 := 0)
      Move(in := 3, out1 => "Boxes".Boxes["CnvF".Sect0.I_RFID_1].V_NumOfDes)
   END_RUNG
   RUNG wire#w1
      P_Trig( "M_Pharmacy_Go_Trig" )
      wire#w2
      "Enqueue3"("Array" := "CnvF".Sect0.V_ArrayBox, Input := "CnvF".Sect0.I_RFID_1, size := "CnvF".Sect0.V_NumOfBox)
   END_RUNG
   RUNG wire#w2
      Sub(in1 := "CnvF".Sect0.V_Busy, in2 := 1, out => "CnvF".Sect0.V_Busy)
   END_RUNG
   RUNG wire#w1
      S_Coil( "M_F_S0_1" )
   END_RUNG
   RUNG wire#w1
      R_Coil( "M_Pharmacy_ChooseRoom" )
   END_RUNG
   // the same network as SCL:
   IF "M_Pharmacy_Go" THEN
       "Boxes".Boxes["CnvF".Sect0.I_RFID_1].V_Destination[1] := "B_Pharmacy_Room1";
       "Boxes".Boxes["CnvF".Sect0.I_RFID_1].V_Completed[1] := "B_Pharmacy_Room1";
       "Boxes".Boxes["CnvF".Sect0.I_RFID_1].V_Destination[2] := "B_Pharmacy_Room2";
       "Boxes".Boxes["CnvF".Sect0.I_RFID_1].V_Completed[2] := "B_Pharmacy_Room2";
       "Boxes".Boxes["CnvF".Sect0.I_RFID_1].V_Destination[3] := "B_Pharmacy_Room3";
       "Boxes".Boxes["CnvF".Sect0.I_RFID_1].V_Completed[3] := "B_Pharmacy_Room3";
       "Boxes".Boxes["CnvF".Sect0.I_RFID_1].V_NumOfComp := 1;
   END_IF;
   IF "M_Pharmacy_Go" AND ("Boxes".Boxes["CnvF".Sect0.I_RFID_2].V_Destination[1] > 0) THEN
       "Boxes".Boxes["CnvF".Sect0.I_RFID_1].V_NumOfDes := 1;
   END_IF;
   IF "M_Pharmacy_Go" AND ("Boxes".Boxes["CnvF".Sect0.I_RFID_1].V_Destination[2] > 0) THEN
       "Boxes".Boxes["CnvF".Sect0.I_RFID_1].V_NumOfDes := 2;
   END_IF;
   IF "M_Pharmacy_Go" AND ("Boxes".Boxes["CnvF".Sect0.I_RFID_1].V_Destination[3] > 0) THEN
       "Boxes".Boxes["CnvF".Sect0.I_RFID_1].V_NumOfDes := 3;
   END_IF;
   #_w1 := "M_Pharmacy_Go" AND NOT "M_Pharmacy_Go_Trig";   // rising edge
   "M_Pharmacy_Go_Trig" := "M_Pharmacy_Go";
   #_w2 := "M_Pharmacy_Go";
   IF #_w1 THEN
       "Enqueue3"("Array" := "CnvF".Sect0.V_ArrayBox,
                  Input := "CnvF".Sect0.I_RFID_1,
                  size := "CnvF".Sect0.V_NumOfBox);
       "CnvF".Sect0.V_Busy := "CnvF".Sect0.V_Busy - 1;
   END_IF;
   IF #_w2 THEN
       "M_F_S0_1" := TRUE;
       "M_Pharmacy_ChooseRoom" := FALSE;
   END_IF;
END_REGION

REGION Network 8: Mode frw sect 0 input
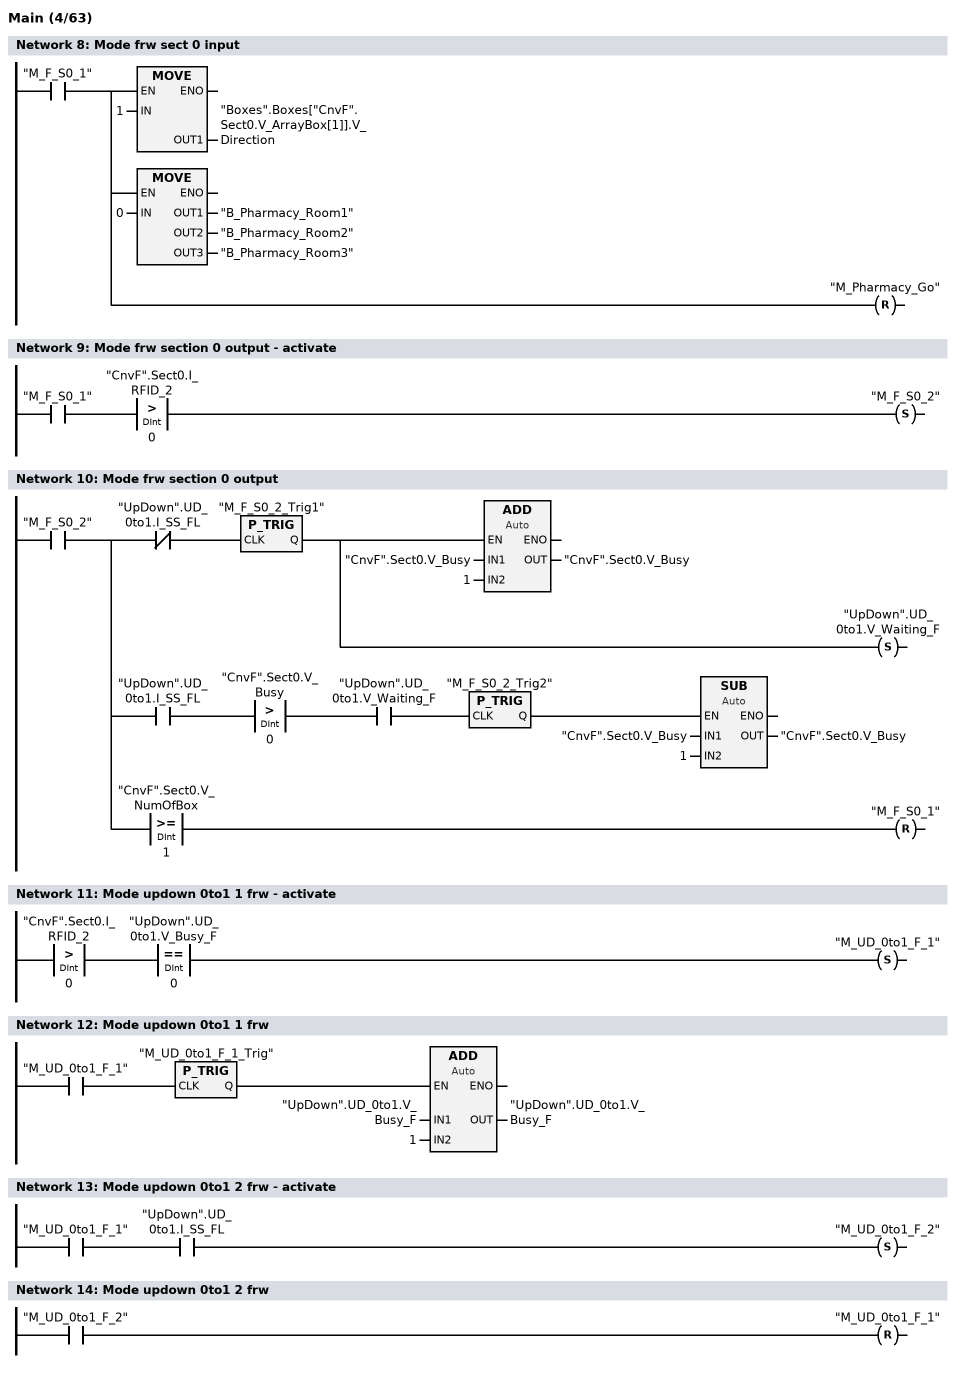
   RUNG wire#powerrail
      Contact( "M_F_S0_1" )
      wire#w1
      Move(in := 1, out1 => "Boxes".Boxes["CnvF".Sect0.V_ArrayBox[1]].V_Direction)
   END_RUNG
   RUNG wire#w1
      Move(in := 0, out1 => "B_Pharmacy_Room1", out2 => "B_Pharmacy_Room2", out3 => "B_Pharmacy_Room3")
   END_RUNG
   RUNG wire#w1
      R_Coil( "M_Pharmacy_Go" )
   END_RUNG
   // the same network as SCL:
   IF "M_F_S0_1" THEN
       "Boxes".Boxes["CnvF".Sect0.V_ArrayBox[1]].V_Direction := 1;
       "B_Pharmacy_Room1" := 0;
       "B_Pharmacy_Room2" := 0;
       "B_Pharmacy_Room3" := 0;
       "M_Pharmacy_Go" := FALSE;
   END_IF;
END_REGION

REGION Network 9: Mode frw section 0 output - activate
   RUNG wire#powerrail
      Contact( "M_F_S0_1" )
      { S7_Templates := "SrcType := DInt" } GT_Contact(in1 := "CnvF".Sect0.I_RFID_2, in2 := 0)
      S_Coil( "M_F_S0_2" )
   END_RUNG
   // the same network as SCL:
   IF "M_F_S0_1" AND ("CnvF".Sect0.I_RFID_2 > 0) THEN "M_F_S0_2" := TRUE; END_IF;
END_REGION

REGION Network 10: Mode frw section 0 output
   RUNG wire#powerrail
      Contact( "M_F_S0_2" )
      wire#w1
      I_Contact( "UpDown".UD_0to1.I_SS_FL )
      P_Trig( "M_F_S0_2_Trig1" )
      wire#w2
      Add(in1 := "CnvF".Sect0.V_Busy, in2 := 1, out => "CnvF".Sect0.V_Busy)
   END_RUNG
   RUNG wire#w2
      S_Coil( "UpDown".UD_0to1.V_Waiting_F )
   END_RUNG
   RUNG wire#w1
      Contact( "UpDown".UD_0to1.I_SS_FL )
      { S7_Templates := "SrcType := DInt" } GT_Contact(in1 := "CnvF".Sect0.V_Busy, in2 := 0)
      Contact( "UpDown".UD_0to1.V_Waiting_F )
      P_Trig( "M_F_S0_2_Trig2" )
      Sub(in1 := "CnvF".Sect0.V_Busy, in2 := 1, out => "CnvF".Sect0.V_Busy)
   END_RUNG
   RUNG wire#w1
      { S7_Templates := "SrcType := DInt" } GE_Contact(in1 := "CnvF".Sect0.V_NumOfBox, in2 := 1)
      R_Coil( "M_F_S0_1" )
   END_RUNG
   // the same network as SCL:
   #_w1 := "M_F_S0_2" AND NOT "UpDown".UD_0to1.I_SS_FL;
   #_w2 := #_w1 AND NOT "M_F_S0_2_Trig1";   // rising edge
   "M_F_S0_2_Trig1" := #_w1;
   IF #_w2 THEN
       "CnvF".Sect0.V_Busy := "CnvF".Sect0.V_Busy + 1;
       "UpDown".UD_0to1.V_Waiting_F := TRUE;
   END_IF;
   #_w3 := "M_F_S0_2" AND "UpDown".UD_0to1.I_SS_FL AND ("CnvF".Sect0.V_Busy > 0) AND "UpDown".UD_0to1.V_Waiting_F;
   #_w4 := #_w3 AND NOT "M_F_S0_2_Trig2";   // rising edge
   "M_F_S0_2_Trig2" := #_w3;
   IF #_w4 THEN "CnvF".Sect0.V_Busy := "CnvF".Sect0.V_Busy - 1; END_IF;
   IF "M_F_S0_2" AND ("CnvF".Sect0.V_NumOfBox >= 1) THEN "M_F_S0_1" := FALSE; END_IF;
END_REGION

REGION Network 11: Mode updown 0to1 1 frw - activate
   RUNG wire#powerrail
      { S7_Templates := "SrcType := DInt" } GT_Contact(in1 := "CnvF".Sect0.I_RFID_2, in2 := 0)
      { S7_Templates := "SrcType := DInt" } EQ_Contact(in1 := "UpDown".UD_0to1.V_Busy_F, in2 := 0)
      S_Coil( "M_UD_0to1_F_1" )
   END_RUNG
   // the same network as SCL:
   IF ("CnvF".Sect0.I_RFID_2 > 0) AND ("UpDown".UD_0to1.V_Busy_F = 0) THEN "M_UD_0to1_F_1" := TRUE; END_IF;
END_REGION

REGION Network 12: Mode updown 0to1 1 frw
   RUNG wire#powerrail
      Contact( "M_UD_0to1_F_1" )
      P_Trig( "M_UD_0to1_F_1_Trig" )
      Add(in1 := "UpDown".UD_0to1.V_Busy_F, in2 := 1, out => "UpDown".UD_0to1.V_Busy_F)
   END_RUNG
   // the same network as SCL:
   #_w1 := "M_UD_0to1_F_1" AND NOT "M_UD_0to1_F_1_Trig";   // rising edge
   "M_UD_0to1_F_1_Trig" := "M_UD_0to1_F_1";
   IF #_w1 THEN "UpDown".UD_0to1.V_Busy_F := "UpDown".UD_0to1.V_Busy_F + 1; END_IF;
END_REGION

REGION Network 13: Mode updown 0to1 2 frw - activate
   RUNG wire#powerrail
      Contact( "M_UD_0to1_F_1" )
      Contact( "UpDown".UD_0to1.I_SS_FL )
      S_Coil( "M_UD_0to1_F_2" )
   END_RUNG
   // the same network as SCL:
   IF "M_UD_0to1_F_1" AND "UpDown".UD_0to1.I_SS_FL THEN "M_UD_0to1_F_2" := TRUE; END_IF;
END_REGION

REGION Network 14: Mode updown 0to1 2 frw
   RUNG wire#powerrail
      Contact( "M_UD_0to1_F_2" )
      R_Coil( "M_UD_0to1_F_1" )
   END_RUNG
   // the same network as SCL:
   IF "M_UD_0to1_F_2" THEN "M_UD_0to1_F_1" := FALSE; END_IF;
END_REGION

REGION Network 15: Mode updown 0to1 3 frw - activate
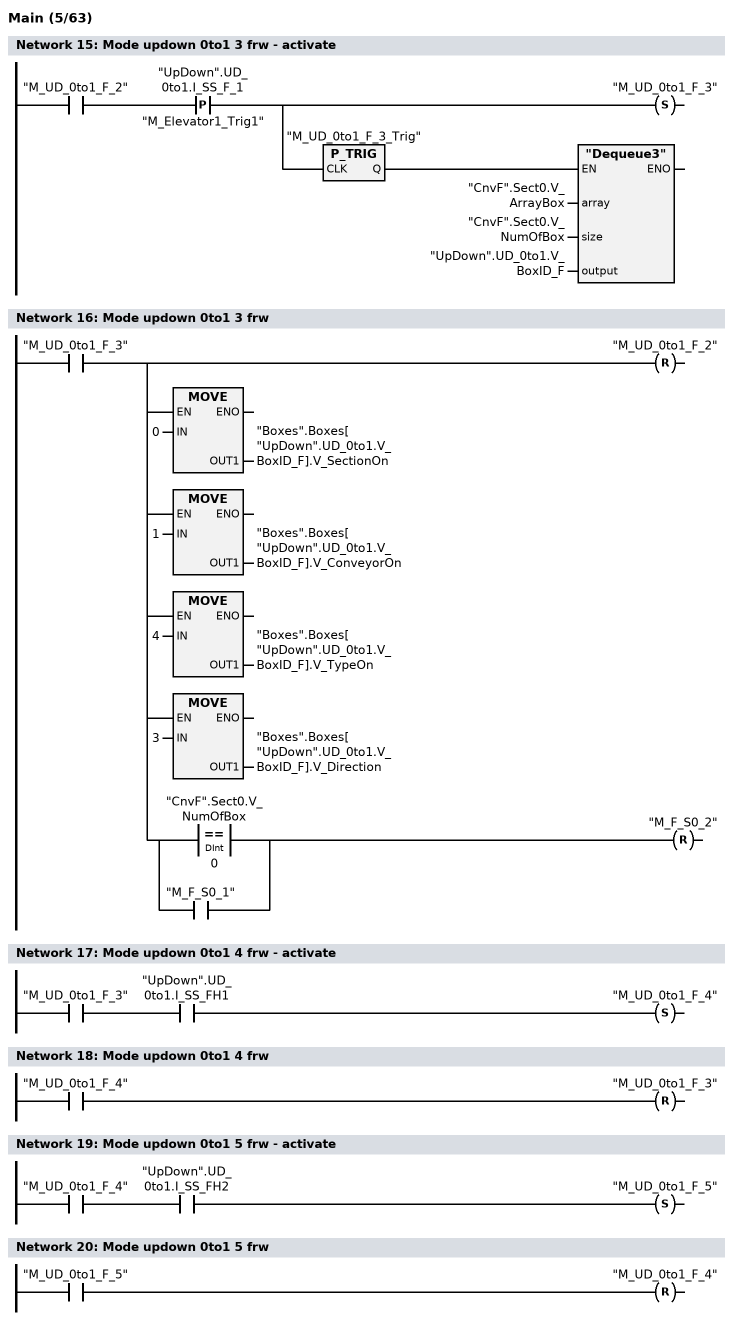
   RUNG wire#powerrail
      Contact( "M_UD_0to1_F_2" )
      P_Contact(operand := "UpDown".UD_0to1.I_SS_F_1, bit := "M_Elevator1_Trig1")
      wire#w1
      S_Coil( "M_UD_0to1_F_3" )
   END_RUNG
   RUNG wire#w1
      P_Trig( "M_UD_0to1_F_3_Trig" )
      "Dequeue3"("array" := "CnvF".Sect0.V_ArrayBox, size := "CnvF".Sect0.V_NumOfBox, output := "UpDown".UD_0to1.V_BoxID_F)
   END_RUNG
   // the same network as SCL:
   #_w1 := "M_UD_0to1_F_2" AND "UpDown".UD_0to1.I_SS_F_1 AND NOT "M_Elevator1_Trig1";   // rising edge of "UpDown".UD_0to1.I_SS_F_1
   "M_Elevator1_Trig1" := "UpDown".UD_0to1.I_SS_F_1;
   IF #_w1 THEN "M_UD_0to1_F_3" := TRUE; END_IF;
   #_w2 := #_w1 AND NOT "M_UD_0to1_F_3_Trig";   // rising edge
   "M_UD_0to1_F_3_Trig" := #_w1;
   IF #_w2 THEN
       "Dequeue3"("array" := "CnvF".Sect0.V_ArrayBox,
                  size := "CnvF".Sect0.V_NumOfBox,
                  output := "UpDown".UD_0to1.V_BoxID_F);
   END_IF;
END_REGION

REGION Network 16: Mode updown 0to1 3 frw
   RUNG wire#powerrail
      Contact( "M_UD_0to1_F_3" )
      wire#w1
      R_Coil( "M_UD_0to1_F_2" )
   END_RUNG
   RUNG wire#w1
      Move(in := 0, out1 => "Boxes".Boxes["UpDown".UD_0to1.V_BoxID_F].V_SectionOn)
   END_RUNG
   RUNG wire#w1
      Move(in := 1, out1 => "Boxes".Boxes["UpDown".UD_0to1.V_BoxID_F].V_ConveyorOn)
   END_RUNG
   RUNG wire#w1
      Move(in := 4, out1 => "Boxes".Boxes["UpDown".UD_0to1.V_BoxID_F].V_TypeOn)
   END_RUNG
   RUNG wire#w1
      Move(in := 3, out1 => "Boxes".Boxes["UpDown".UD_0to1.V_BoxID_F].V_Direction)
   END_RUNG
   RUNG wire#w1
      { S7_Templates := "SrcType := DInt" } EQ_Contact(in1 := "CnvF".Sect0.V_NumOfBox, in2 := 0)
      wire#w2
      R_Coil( "M_F_S0_2" )
   END_RUNG
   RUNG wire#w1
      Contact( "M_F_S0_1" )
   END_RUNG wire#w2
   // the same network as SCL:
   IF "M_UD_0to1_F_3" THEN
       "M_UD_0to1_F_2" := FALSE;
       "Boxes".Boxes["UpDown".UD_0to1.V_BoxID_F].V_SectionOn := 0;
       "Boxes".Boxes["UpDown".UD_0to1.V_BoxID_F].V_ConveyorOn := 1;
       "Boxes".Boxes["UpDown".UD_0to1.V_BoxID_F].V_TypeOn := 4;
       "Boxes".Boxes["UpDown".UD_0to1.V_BoxID_F].V_Direction := 3;
   END_IF;
   IF "M_UD_0to1_F_3" AND (("CnvF".Sect0.V_NumOfBox = 0) OR "M_F_S0_1") THEN "M_F_S0_2" := FALSE; END_IF;
END_REGION

REGION Network 17: Mode updown 0to1 4 frw - activate
   RUNG wire#powerrail
      Contact( "M_UD_0to1_F_3" )
      Contact( "UpDown".UD_0to1.I_SS_FH1 )
      S_Coil( "M_UD_0to1_F_4" )
   END_RUNG
   // the same network as SCL:
   IF "M_UD_0to1_F_3" AND "UpDown".UD_0to1.I_SS_FH1 THEN "M_UD_0to1_F_4" := TRUE; END_IF;
END_REGION

REGION Network 18: Mode updown 0to1 4 frw
   RUNG wire#powerrail
      Contact( "M_UD_0to1_F_4" )
      R_Coil( "M_UD_0to1_F_3" )
   END_RUNG
   // the same network as SCL:
   IF "M_UD_0to1_F_4" THEN "M_UD_0to1_F_3" := FALSE; END_IF;
END_REGION

REGION Network 19: Mode updown 0to1 5 frw - activate
   RUNG wire#powerrail
      Contact( "M_UD_0to1_F_4" )
      Contact( "UpDown".UD_0to1.I_SS_FH2 )
      S_Coil( "M_UD_0to1_F_5" )
   END_RUNG
   // the same network as SCL:
   IF "M_UD_0to1_F_4" AND "UpDown".UD_0to1.I_SS_FH2 THEN "M_UD_0to1_F_5" := TRUE; END_IF;
END_REGION

REGION Network 20: Mode updown 0to1 5 frw
   RUNG wire#powerrail
      Contact( "M_UD_0to1_F_5" )
      R_Coil( "M_UD_0to1_F_4" )
   END_RUNG
   // the same network as SCL:
   IF "M_UD_0to1_F_5" THEN "M_UD_0to1_F_4" := FALSE; END_IF;
END_REGION

REGION Network 21: Mode updown 0to1 6 frw - activate
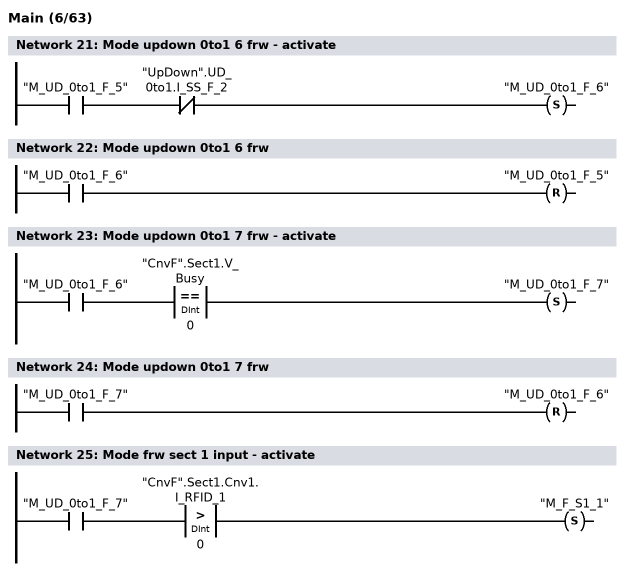
   RUNG wire#powerrail
      Contact( "M_UD_0to1_F_5" )
      I_Contact( "UpDown".UD_0to1.I_SS_F_2 )
      S_Coil( "M_UD_0to1_F_6" )
   END_RUNG
   // the same network as SCL:
   IF "M_UD_0to1_F_5" AND NOT "UpDown".UD_0to1.I_SS_F_2 THEN "M_UD_0to1_F_6" := TRUE; END_IF;
END_REGION

REGION Network 22: Mode updown 0to1 6 frw
   RUNG wire#powerrail
      Contact( "M_UD_0to1_F_6" )
      R_Coil( "M_UD_0to1_F_5" )
   END_RUNG
   // the same network as SCL:
   IF "M_UD_0to1_F_6" THEN "M_UD_0to1_F_5" := FALSE; END_IF;
END_REGION

REGION Network 23: Mode updown 0to1 7 frw - activate
   RUNG wire#powerrail
      Contact( "M_UD_0to1_F_6" )
      { S7_Templates := "SrcType := DInt" } EQ_Contact(in1 := "CnvF".Sect1.V_Busy, in2 := 0)
      S_Coil( "M_UD_0to1_F_7" )
   END_RUNG
   // the same network as SCL:
   IF "M_UD_0to1_F_6" AND ("CnvF".Sect1.V_Busy = 0) THEN "M_UD_0to1_F_7" := TRUE; END_IF;
END_REGION

REGION Network 24: Mode updown 0to1 7 frw
   RUNG wire#powerrail
      Contact( "M_UD_0to1_F_7" )
      R_Coil( "M_UD_0to1_F_6" )
   END_RUNG
   // the same network as SCL:
   IF "M_UD_0to1_F_7" THEN "M_UD_0to1_F_6" := FALSE; END_IF;
END_REGION

REGION Network 25: Mode frw sect 1 input - activate
   RUNG wire#powerrail
      Contact( "M_UD_0to1_F_7" )
      { S7_Templates := "SrcType := DInt" } GT_Contact(in1 := "CnvF".Sect1.Cnv1.I_RFID_1, in2 := 0)
      S_Coil( "M_F_S1_1" )
   END_RUNG
   // the same network as SCL:
   IF "M_UD_0to1_F_7" AND ("CnvF".Sect1.Cnv1.I_RFID_1 > 0) THEN "M_F_S1_1" := TRUE; END_IF;
END_REGION

REGION Network 26: Mode frw sect 1 input
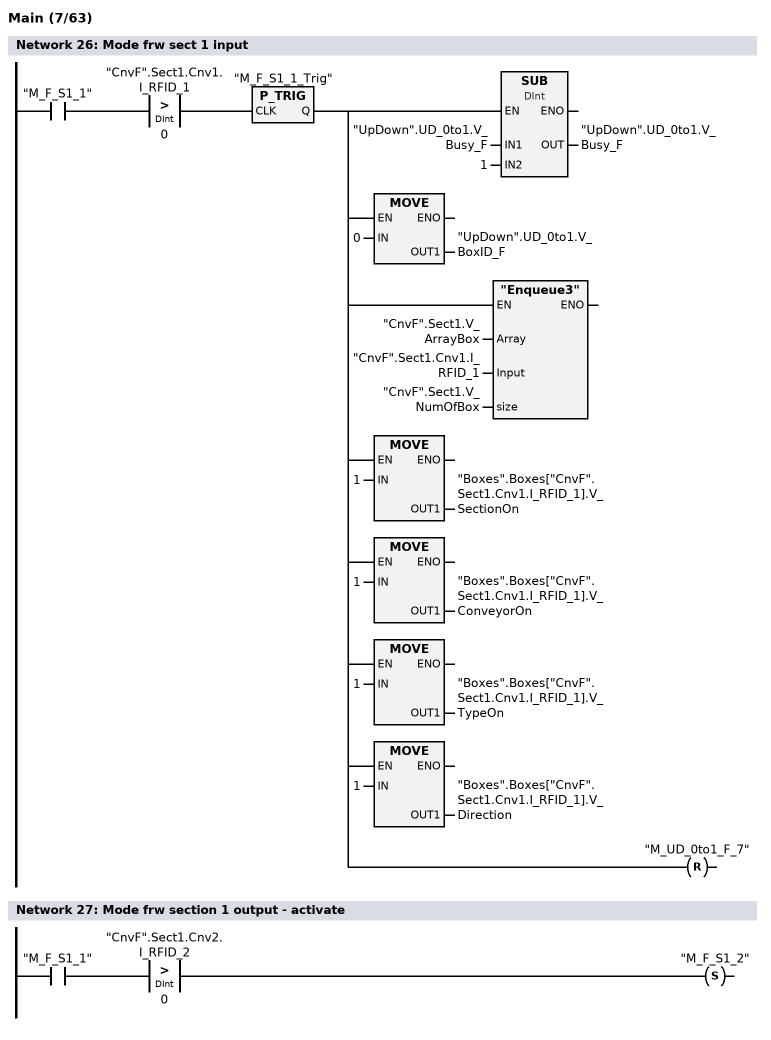
   RUNG wire#powerrail
      Contact( "M_F_S1_1" )
      { S7_Templates := "SrcType := DInt" } GT_Contact(in1 := "CnvF".Sect1.Cnv1.I_RFID_1, in2 := 0)
      P_Trig( "M_F_S1_1_Trig" )
      wire#w1
      { S7_Templates := "SrcType := DInt" } Sub(in1 := "UpDown".UD_0to1.V_Busy_F, in2 := 1, out => "UpDown".UD_0to1.V_Busy_F)
   END_RUNG
   RUNG wire#w1
      Move(in := 0, out1 => "UpDown".UD_0to1.V_BoxID_F)
   END_RUNG
   RUNG wire#w1
      "Enqueue3"("Array" := "CnvF".Sect1.V_ArrayBox, Input := "CnvF".Sect1.Cnv1.I_RFID_1, size := "CnvF".Sect1.V_NumOfBox)
   END_RUNG
   RUNG wire#w1
      Move(in := 1, out1 => "Boxes".Boxes["CnvF".Sect1.Cnv1.I_RFID_1].V_SectionOn)
   END_RUNG
   RUNG wire#w1
      Move(in := 1, out1 => "Boxes".Boxes["CnvF".Sect1.Cnv1.I_RFID_1].V_ConveyorOn)
   END_RUNG
   RUNG wire#w1
      Move(in := 1, out1 => "Boxes".Boxes["CnvF".Sect1.Cnv1.I_RFID_1].V_TypeOn)
   END_RUNG
   RUNG wire#w1
      Move(in := 1, out1 => "Boxes".Boxes["CnvF".Sect1.Cnv1.I_RFID_1].V_Direction)
   END_RUNG
   RUNG wire#w1
      R_Coil( "M_UD_0to1_F_7" )
   END_RUNG
   // the same network as SCL:
   #_w1 := "M_F_S1_1" AND ("CnvF".Sect1.Cnv1.I_RFID_1 > 0);
   #_w2 := #_w1 AND NOT "M_F_S1_1_Trig";   // rising edge
   "M_F_S1_1_Trig" := #_w1;
   IF #_w2 THEN
       "UpDown".UD_0to1.V_Busy_F := "UpDown".UD_0to1.V_Busy_F - 1;
       "UpDown".UD_0to1.V_BoxID_F := 0;
       "Enqueue3"("Array" := "CnvF".Sect1.V_ArrayBox,
                  Input := "CnvF".Sect1.Cnv1.I_RFID_1,
                  size := "CnvF".Sect1.V_NumOfBox);
       "Boxes".Boxes["CnvF".Sect1.Cnv1.I_RFID_1].V_SectionOn := 1;
       "Boxes".Boxes["CnvF".Sect1.Cnv1.I_RFID_1].V_ConveyorOn := 1;
       "Boxes".Boxes["CnvF".Sect1.Cnv1.I_RFID_1].V_TypeOn := 1;
       "Boxes".Boxes["CnvF".Sect1.Cnv1.I_RFID_1].V_Direction := 1;
       "M_UD_0to1_F_7" := FALSE;
   END_IF;
END_REGION

REGION Network 27: Mode frw section 1 output - activate
   RUNG wire#powerrail
      Contact( "M_F_S1_1" )
      { S7_Templates := "SrcType := DInt" } GT_Contact(in1 := "CnvF".Sect1.Cnv2.I_RFID_2, in2 := 0)
      S_Coil( "M_F_S1_2" )
   END_RUNG
   // the same network as SCL:
   IF "M_F_S1_1" AND ("CnvF".Sect1.Cnv2.I_RFID_2 > 0) THEN "M_F_S1_2" := TRUE; END_IF;
END_REGION

REGION Network 28: Mode frw section 1 output
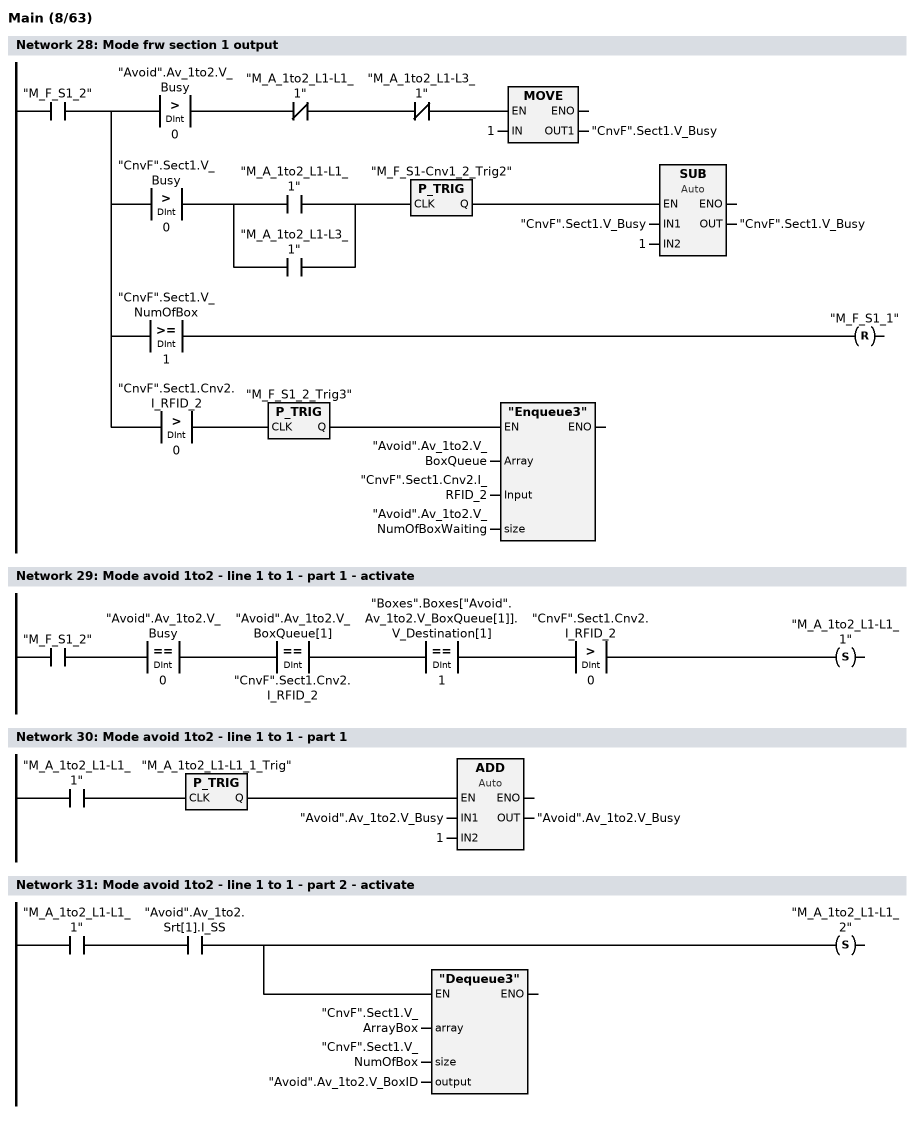
   RUNG wire#powerrail
      Contact( "M_F_S1_2" )
      wire#w1
      { S7_Templates := "SrcType := DInt" } GT_Contact(in1 := "Avoid".Av_1to2.V_Busy, in2 := 0)
      I_Contact( "M_A_1to2_L1-L1_1" )
      I_Contact( "M_A_1to2_L1-L3_1" )
      Move(in := 1, out1 => "CnvF".Sect1.V_Busy)
   END_RUNG
   RUNG wire#w1
      { S7_Templates := "SrcType := DInt" } GT_Contact(in1 := "CnvF".Sect1.V_Busy, in2 := 0)
      wire#w2
      Contact( "M_A_1to2_L1-L1_1" )
      wire#w3
      P_Trig( "M_F_S1-Cnv1_2_Trig2" )
      Sub(in1 := "CnvF".Sect1.V_Busy, in2 := 1, out => "CnvF".Sect1.V_Busy)
   END_RUNG
   RUNG wire#w2
      Contact( "M_A_1to2_L1-L3_1" )
   END_RUNG wire#w3
   RUNG wire#w1
      { S7_Templates := "SrcType := DInt" } GE_Contact(in1 := "CnvF".Sect1.V_NumOfBox, in2 := 1)
      R_Coil( "M_F_S1_1" )
   END_RUNG
   RUNG wire#w1
      { S7_Templates := "SrcType := DInt" } GT_Contact(in1 := "CnvF".Sect1.Cnv2.I_RFID_2, in2 := 0)
      P_Trig( "M_F_S1_2_Trig3" )
      "Enqueue3"("Array" := "Avoid".Av_1to2.V_BoxQueue, Input := "CnvF".Sect1.Cnv2.I_RFID_2, size := "Avoid".Av_1to2.V_NumOfBoxWaiting)
   END_RUNG
   // the same network as SCL:
   IF "M_F_S1_2" AND ("Avoid".Av_1to2.V_Busy > 0) AND NOT "M_A_1to2_L1-L1_1" AND NOT "M_A_1to2_L1-L3_1" THEN
       "CnvF".Sect1.V_Busy := 1;
   END_IF;
   #_w1 := "M_F_S1_2" AND ("CnvF".Sect1.V_Busy > 0) AND ("M_A_1to2_L1-L1_1" OR "M_A_1to2_L1-L3_1");
   #_w2 := #_w1 AND NOT "M_F_S1-Cnv1_2_Trig2";   // rising edge
   "M_F_S1-Cnv1_2_Trig2" := #_w1;
   IF #_w2 THEN "CnvF".Sect1.V_Busy := "CnvF".Sect1.V_Busy - 1; END_IF;
   IF "M_F_S1_2" AND ("CnvF".Sect1.V_NumOfBox >= 1) THEN "M_F_S1_1" := FALSE; END_IF;
   #_w3 := "M_F_S1_2" AND ("CnvF".Sect1.Cnv2.I_RFID_2 > 0);
   #_w4 := #_w3 AND NOT "M_F_S1_2_Trig3";   // rising edge
   "M_F_S1_2_Trig3" := #_w3;
   IF #_w4 THEN
       "Enqueue3"("Array" := "Avoid".Av_1to2.V_BoxQueue,
                  Input := "CnvF".Sect1.Cnv2.I_RFID_2,
                  size := "Avoid".Av_1to2.V_NumOfBoxWaiting);
   END_IF;
END_REGION

REGION Network 29: Mode avoid 1to2 - line 1 to 1 - part 1 - activate
   RUNG wire#powerrail
      Contact( "M_F_S1_2" )
      { S7_Templates := "SrcType := DInt" } EQ_Contact(in1 := "Avoid".Av_1to2.V_Busy, in2 := 0)
      { S7_Templates := "SrcType := DInt" } EQ_Contact(in1 := "Avoid".Av_1to2.V_BoxQueue[1], in2 := "CnvF".Sect1.Cnv2.I_RFID_2)
      { S7_Templates := "SrcType := DInt" } EQ_Contact(in1 := "Boxes".Boxes["Avoid".Av_1to2.V_BoxQueue[1]].V_Destination[1], in2 := 1)
      { S7_Templates := "SrcType := DInt" } GT_Contact(in1 := "CnvF".Sect1.Cnv2.I_RFID_2, in2 := 0)
      S_Coil( "M_A_1to2_L1-L1_1" )
   END_RUNG
   // the same network as SCL:
   IF "M_F_S1_2" AND ("Avoid".Av_1to2.V_Busy = 0) AND ("Avoid".Av_1to2.V_BoxQueue[1] = "CnvF".Sect1.Cnv2.I_RFID_2) AND ("Boxes".Boxes["Avoid".Av_1to2.V_BoxQueue[1]].V_Destination[1] = 1) AND ("CnvF".Sect1.Cnv2.I_RFID_2 > 0) THEN
       "M_A_1to2_L1-L1_1" := TRUE;
   END_IF;
END_REGION

REGION Network 30: Mode avoid 1to2 - line 1 to 1 - part 1
   RUNG wire#powerrail
      Contact( "M_A_1to2_L1-L1_1" )
      P_Trig( "M_A_1to2_L1-L1_1_Trig" )
      Add(in1 := "Avoid".Av_1to2.V_Busy, in2 := 1, out => "Avoid".Av_1to2.V_Busy)
   END_RUNG
   // the same network as SCL:
   #_w1 := "M_A_1to2_L1-L1_1" AND NOT "M_A_1to2_L1-L1_1_Trig";   // rising edge
   "M_A_1to2_L1-L1_1_Trig" := "M_A_1to2_L1-L1_1";
   IF #_w1 THEN "Avoid".Av_1to2.V_Busy := "Avoid".Av_1to2.V_Busy + 1; END_IF;
END_REGION

REGION Network 31: Mode avoid 1to2 - line 1 to 1 - part 2 - activate
   RUNG wire#powerrail
      Contact( "M_A_1to2_L1-L1_1" )
      Contact( "Avoid".Av_1to2.Srt[1].I_SS )
      wire#w1
      S_Coil( "M_A_1to2_L1-L1_2" )
   END_RUNG
   RUNG wire#w1
      "Dequeue3"("array" := "CnvF".Sect1.V_ArrayBox, size := "CnvF".Sect1.V_NumOfBox, output := "Avoid".Av_1to2.V_BoxID)
   END_RUNG
   // the same network as SCL:
   IF "M_A_1to2_L1-L1_1" AND "Avoid".Av_1to2.Srt[1].I_SS THEN
       "M_A_1to2_L1-L1_2" := TRUE;
       "Dequeue3"("array" := "CnvF".Sect1.V_ArrayBox,
                  size := "CnvF".Sect1.V_NumOfBox,
                  output := "Avoid".Av_1to2.V_BoxID);
   END_IF;
END_REGION

REGION Network 32: Mode avoid 1to2 - line 1 to 1 - part 2
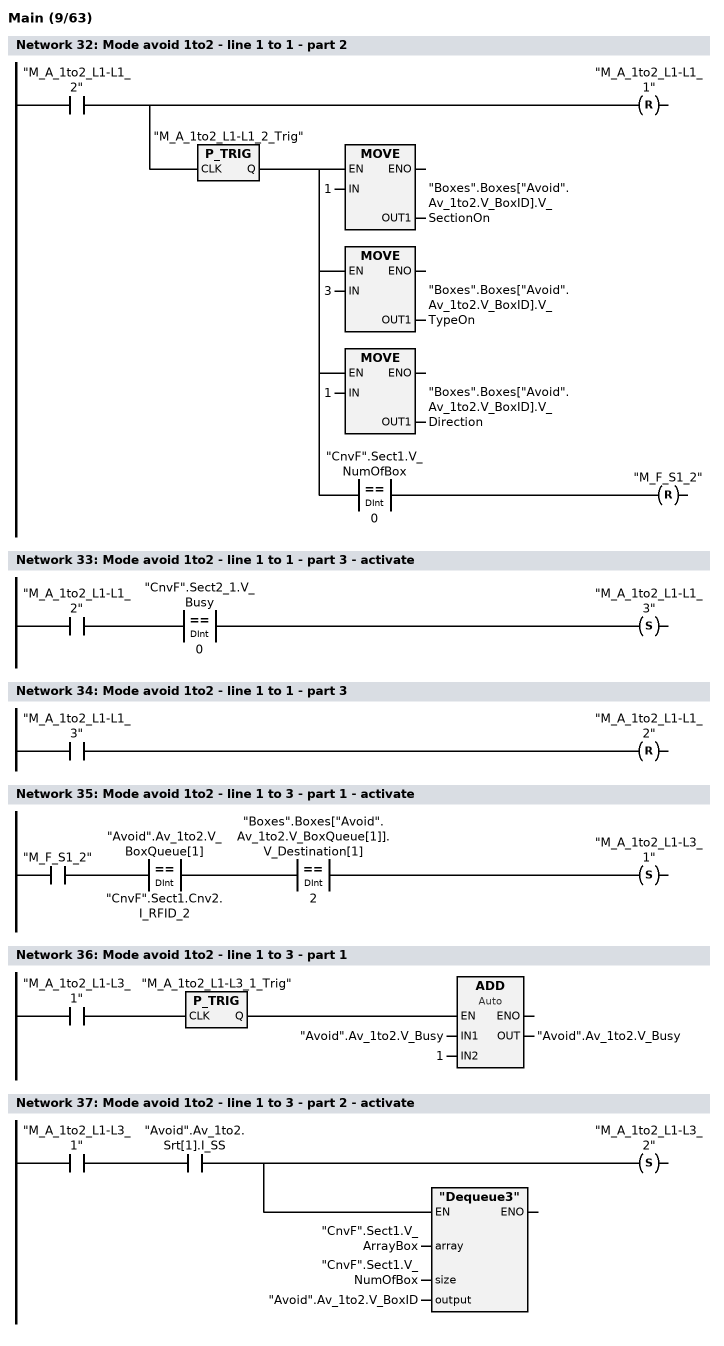
   RUNG wire#powerrail
      Contact( "M_A_1to2_L1-L1_2" )
      wire#w1
      R_Coil( "M_A_1to2_L1-L1_1" )
   END_RUNG
   RUNG wire#w1
      P_Trig( "M_A_1to2_L1-L1_2_Trig" )
      wire#w2
      Move(in := 1, out1 => "Boxes".Boxes["Avoid".Av_1to2.V_BoxID].V_SectionOn)
   END_RUNG
   RUNG wire#w2
      Move(in := 3, out1 => "Boxes".Boxes["Avoid".Av_1to2.V_BoxID].V_TypeOn)
   END_RUNG
   RUNG wire#w2
      Move(in := 1, out1 => "Boxes".Boxes["Avoid".Av_1to2.V_BoxID].V_Direction)
   END_RUNG
   RUNG wire#w2
      { S7_Templates := "SrcType := DInt" } EQ_Contact(in1 := "CnvF".Sect1.V_NumOfBox, in2 := 0)
      R_Coil( "M_F_S1_2" )
   END_RUNG
   // the same network as SCL:
   IF "M_A_1to2_L1-L1_2" THEN "M_A_1to2_L1-L1_1" := FALSE; END_IF;
   #_w1 := "M_A_1to2_L1-L1_2" AND NOT "M_A_1to2_L1-L1_2_Trig";   // rising edge
   "M_A_1to2_L1-L1_2_Trig" := "M_A_1to2_L1-L1_2";
   IF #_w1 THEN
       "Boxes".Boxes["Avoid".Av_1to2.V_BoxID].V_SectionOn := 1;
       "Boxes".Boxes["Avoid".Av_1to2.V_BoxID].V_TypeOn := 3;
       "Boxes".Boxes["Avoid".Av_1to2.V_BoxID].V_Direction := 1;
   END_IF;
   IF #_w1 AND ("CnvF".Sect1.V_NumOfBox = 0) THEN "M_F_S1_2" := FALSE; END_IF;
END_REGION

REGION Network 33: Mode avoid 1to2 - line 1 to 1 - part 3 - activate
   RUNG wire#powerrail
      Contact( "M_A_1to2_L1-L1_2" )
      { S7_Templates := "SrcType := DInt" } EQ_Contact(in1 := "CnvF".Sect2_1.V_Busy, in2 := 0)
      S_Coil( "M_A_1to2_L1-L1_3" )
   END_RUNG
   // the same network as SCL:
   IF "M_A_1to2_L1-L1_2" AND ("CnvF".Sect2_1.V_Busy = 0) THEN "M_A_1to2_L1-L1_3" := TRUE; END_IF;
END_REGION

REGION Network 34: Mode avoid 1to2 - line 1 to 1 - part 3
   RUNG wire#powerrail
      Contact( "M_A_1to2_L1-L1_3" )
      R_Coil( "M_A_1to2_L1-L1_2" )
   END_RUNG
   // the same network as SCL:
   IF "M_A_1to2_L1-L1_3" THEN "M_A_1to2_L1-L1_2" := FALSE; END_IF;
END_REGION

REGION Network 35: Mode avoid 1to2 - line 1 to 3 - part 1 - activate
   RUNG wire#powerrail
      Contact( "M_F_S1_2" )
      { S7_Templates := "SrcType := DInt" } EQ_Contact(in1 := "Avoid".Av_1to2.V_BoxQueue[1], in2 := "CnvF".Sect1.Cnv2.I_RFID_2)
      { S7_Templates := "SrcType := DInt" } EQ_Contact(in1 := "Boxes".Boxes["Avoid".Av_1to2.V_BoxQueue[1]].V_Destination[1], in2 := 2)
      S_Coil( "M_A_1to2_L1-L3_1" )
   END_RUNG
   // the same network as SCL:
   IF "M_F_S1_2" AND ("Avoid".Av_1to2.V_BoxQueue[1] = "CnvF".Sect1.Cnv2.I_RFID_2) AND ("Boxes".Boxes["Avoid".Av_1to2.V_BoxQueue[1]].V_Destination[1] = 2) THEN
       "M_A_1to2_L1-L3_1" := TRUE;
   END_IF;
END_REGION

REGION Network 36: Mode avoid 1to2 - line 1 to 3 - part 1
   RUNG wire#powerrail
      Contact( "M_A_1to2_L1-L3_1" )
      P_Trig( "M_A_1to2_L1-L3_1_Trig" )
      Add(in1 := "Avoid".Av_1to2.V_Busy, in2 := 1, out => "Avoid".Av_1to2.V_Busy)
   END_RUNG
   // the same network as SCL:
   #_w1 := "M_A_1to2_L1-L3_1" AND NOT "M_A_1to2_L1-L3_1_Trig";   // rising edge
   "M_A_1to2_L1-L3_1_Trig" := "M_A_1to2_L1-L3_1";
   IF #_w1 THEN "Avoid".Av_1to2.V_Busy := "Avoid".Av_1to2.V_Busy + 1; END_IF;
END_REGION

REGION Network 37: Mode avoid 1to2 - line 1 to 3 - part 2 - activate
   RUNG wire#powerrail
      Contact( "M_A_1to2_L1-L3_1" )
      Contact( "Avoid".Av_1to2.Srt[1].I_SS )
      wire#w1
      S_Coil( "M_A_1to2_L1-L3_2" )
   END_RUNG
   RUNG wire#w1
      "Dequeue3"("array" := "CnvF".Sect1.V_ArrayBox, size := "CnvF".Sect1.V_NumOfBox, output := "Avoid".Av_1to2.V_BoxID)
   END_RUNG
   // the same network as SCL:
   IF "M_A_1to2_L1-L3_1" AND "Avoid".Av_1to2.Srt[1].I_SS THEN
       "M_A_1to2_L1-L3_2" := TRUE;
       "Dequeue3"("array" := "CnvF".Sect1.V_ArrayBox,
                  size := "CnvF".Sect1.V_NumOfBox,
                  output := "Avoid".Av_1to2.V_BoxID);
   END_IF;
END_REGION

REGION Network 38: Mode avoid 1to2 - line 1 to 3 - part 2
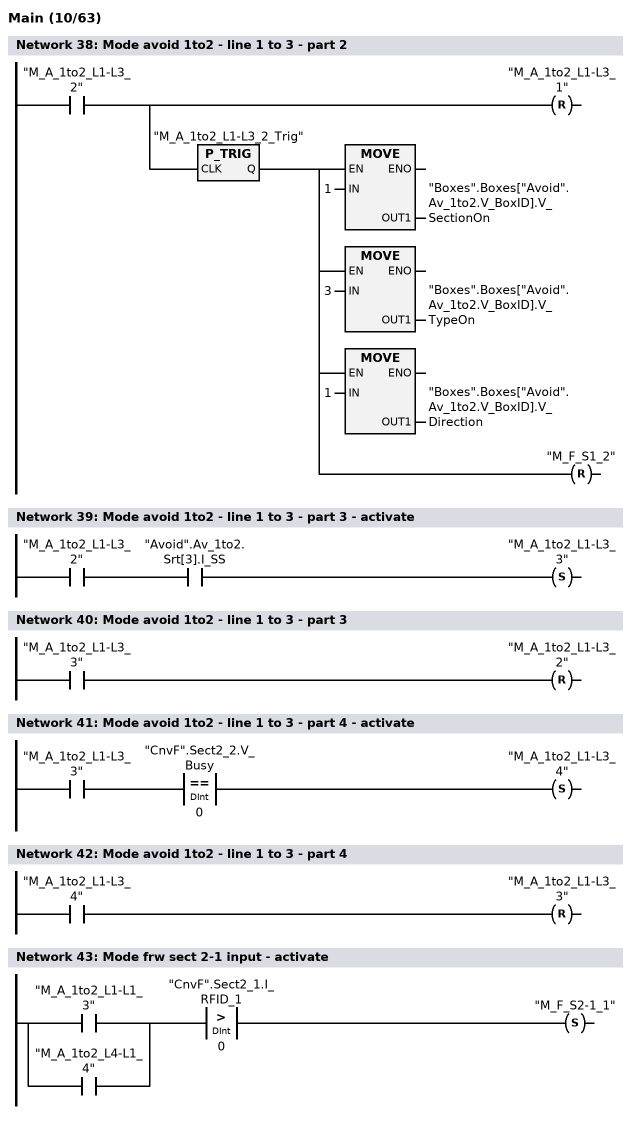
   RUNG wire#powerrail
      Contact( "M_A_1to2_L1-L3_2" )
      wire#w1
      R_Coil( "M_A_1to2_L1-L3_1" )
   END_RUNG
   RUNG wire#w1
      P_Trig( "M_A_1to2_L1-L3_2_Trig" )
      wire#w2
      Move(in := 1, out1 => "Boxes".Boxes["Avoid".Av_1to2.V_BoxID].V_SectionOn)
   END_RUNG
   RUNG wire#w2
      Move(in := 3, out1 => "Boxes".Boxes["Avoid".Av_1to2.V_BoxID].V_TypeOn)
   END_RUNG
   RUNG wire#w2
      Move(in := 1, out1 => "Boxes".Boxes["Avoid".Av_1to2.V_BoxID].V_Direction)
   END_RUNG
   RUNG wire#w2
      R_Coil( "M_F_S1_2" )
   END_RUNG
   // the same network as SCL:
   IF "M_A_1to2_L1-L3_2" THEN "M_A_1to2_L1-L3_1" := FALSE; END_IF;
   #_w1 := "M_A_1to2_L1-L3_2" AND NOT "M_A_1to2_L1-L3_2_Trig";   // rising edge
   "M_A_1to2_L1-L3_2_Trig" := "M_A_1to2_L1-L3_2";
   IF #_w1 THEN
       "Boxes".Boxes["Avoid".Av_1to2.V_BoxID].V_SectionOn := 1;
       "Boxes".Boxes["Avoid".Av_1to2.V_BoxID].V_TypeOn := 3;
       "Boxes".Boxes["Avoid".Av_1to2.V_BoxID].V_Direction := 1;
       "M_F_S1_2" := FALSE;
   END_IF;
END_REGION

REGION Network 39: Mode avoid 1to2 - line 1 to 3 - part 3 - activate
   RUNG wire#powerrail
      Contact( "M_A_1to2_L1-L3_2" )
      Contact( "Avoid".Av_1to2.Srt[3].I_SS )
      S_Coil( "M_A_1to2_L1-L3_3" )
   END_RUNG
   // the same network as SCL:
   IF "M_A_1to2_L1-L3_2" AND "Avoid".Av_1to2.Srt[3].I_SS THEN "M_A_1to2_L1-L3_3" := TRUE; END_IF;
END_REGION

REGION Network 40: Mode avoid 1to2 - line 1 to 3 - part 3
   RUNG wire#powerrail
      Contact( "M_A_1to2_L1-L3_3" )
      R_Coil( "M_A_1to2_L1-L3_2" )
   END_RUNG
   // the same network as SCL:
   IF "M_A_1to2_L1-L3_3" THEN "M_A_1to2_L1-L3_2" := FALSE; END_IF;
END_REGION

REGION Network 41: Mode avoid 1to2 - line 1 to 3 - part 4 - activate
   RUNG wire#powerrail
      Contact( "M_A_1to2_L1-L3_3" )
      { S7_Templates := "SrcType := DInt" } EQ_Contact(in1 := "CnvF".Sect2_2.V_Busy, in2 := 0)
      S_Coil( "M_A_1to2_L1-L3_4" )
   END_RUNG
   // the same network as SCL:
   IF "M_A_1to2_L1-L3_3" AND ("CnvF".Sect2_2.V_Busy = 0) THEN "M_A_1to2_L1-L3_4" := TRUE; END_IF;
END_REGION

REGION Network 42: Mode avoid 1to2 - line 1 to 3 - part 4
   RUNG wire#powerrail
      Contact( "M_A_1to2_L1-L3_4" )
      R_Coil( "M_A_1to2_L1-L3_3" )
   END_RUNG
   // the same network as SCL:
   IF "M_A_1to2_L1-L3_4" THEN "M_A_1to2_L1-L3_3" := FALSE; END_IF;
END_REGION

REGION Network 43: Mode frw sect 2-1 input - activate
   RUNG wire#powerrail
      Contact( "M_A_1to2_L1-L1_3" )
      wire#w1
      { S7_Templates := "SrcType := DInt" } GT_Contact(in1 := "CnvF".Sect2_1.I_RFID_1, in2 := 0)
      S_Coil( "M_F_S2-1_1" )
   END_RUNG
   RUNG wire#powerrail
      Contact( "M_A_1to2_L4-L1_4" )
   END_RUNG wire#w1
   // the same network as SCL:
   IF ("M_A_1to2_L1-L1_3" OR "M_A_1to2_L4-L1_4") AND ("CnvF".Sect2_1.I_RFID_1 > 0) THEN
       "M_F_S2-1_1" := TRUE;
   END_IF;
END_REGION

REGION Network 44: Mode frw sect 2-1 input
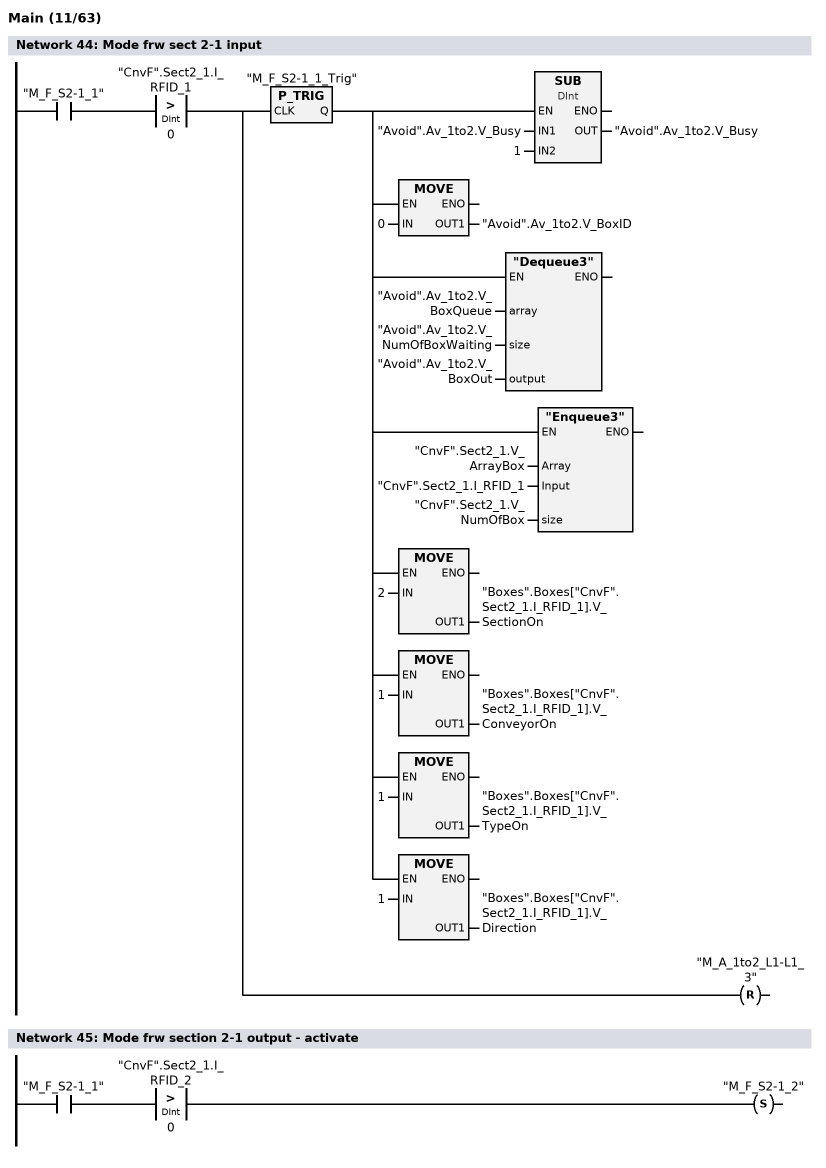
   RUNG wire#powerrail
      Contact( "M_F_S2-1_1" )
      { S7_Templates := "SrcType := DInt" } GT_Contact(in1 := "CnvF".Sect2_1.I_RFID_1, in2 := 0)
      wire#w1
      P_Trig( "M_F_S2-1_1_Trig" )
      wire#w2
      { S7_Templates := "SrcType := DInt" } Sub(in1 := "Avoid".Av_1to2.V_Busy, in2 := 1, out => "Avoid".Av_1to2.V_Busy)
   END_RUNG
   RUNG wire#w2
      Move(in := 0, out1 => "Avoid".Av_1to2.V_BoxID)
   END_RUNG
   RUNG wire#w2
      "Dequeue3"("array" := "Avoid".Av_1to2.V_BoxQueue, size := "Avoid".Av_1to2.V_NumOfBoxWaiting, output := "Avoid".Av_1to2.V_BoxOut)
   END_RUNG
   RUNG wire#w2
      "Enqueue3"("Array" := "CnvF".Sect2_1.V_ArrayBox, Input := "CnvF".Sect2_1.I_RFID_1, size := "CnvF".Sect2_1.V_NumOfBox)
   END_RUNG
   RUNG wire#w2
      Move(in := 2, out1 => "Boxes".Boxes["CnvF".Sect2_1.I_RFID_1].V_SectionOn)
   END_RUNG
   RUNG wire#w2
      Move(in := 1, out1 => "Boxes".Boxes["CnvF".Sect2_1.I_RFID_1].V_ConveyorOn)
   END_RUNG
   RUNG wire#w2
      Move(in := 1, out1 => "Boxes".Boxes["CnvF".Sect2_1.I_RFID_1].V_TypeOn)
   END_RUNG
   RUNG wire#w2
      Move(in := 1, out1 => "Boxes".Boxes["CnvF".Sect2_1.I_RFID_1].V_Direction)
   END_RUNG
   RUNG wire#w1
      R_Coil( "M_A_1to2_L1-L1_3" )
   END_RUNG
   // the same network as SCL:
   #_w1 := "M_F_S2-1_1" AND ("CnvF".Sect2_1.I_RFID_1 > 0);
   #_w2 := #_w1 AND NOT "M_F_S2-1_1_Trig";   // rising edge
   "M_F_S2-1_1_Trig" := #_w1;
   IF #_w2 THEN
       "Avoid".Av_1to2.V_Busy := "Avoid".Av_1to2.V_Busy - 1;
       "Avoid".Av_1to2.V_BoxID := 0;
       "Dequeue3"("array" := "Avoid".Av_1to2.V_BoxQueue,
                  size := "Avoid".Av_1to2.V_NumOfBoxWaiting,
                  output := "Avoid".Av_1to2.V_BoxOut);
       "Enqueue3"("Array" := "CnvF".Sect2_1.V_ArrayBox,
                  Input := "CnvF".Sect2_1.I_RFID_1,
                  size := "CnvF".Sect2_1.V_NumOfBox);
       "Boxes".Boxes["CnvF".Sect2_1.I_RFID_1].V_SectionOn := 2;
       "Boxes".Boxes["CnvF".Sect2_1.I_RFID_1].V_ConveyorOn := 1;
       "Boxes".Boxes["CnvF".Sect2_1.I_RFID_1].V_TypeOn := 1;
       "Boxes".Boxes["CnvF".Sect2_1.I_RFID_1].V_Direction := 1;
   END_IF;
   IF #_w1 THEN "M_A_1to2_L1-L1_3" := FALSE; END_IF;
END_REGION

REGION Network 45: Mode frw section 2-1 output - activate
   RUNG wire#powerrail
      Contact( "M_F_S2-1_1" )
      { S7_Templates := "SrcType := DInt" } GT_Contact(in1 := "CnvF".Sect2_1.I_RFID_2, in2 := 0)
      S_Coil( "M_F_S2-1_2" )
   END_RUNG
   // the same network as SCL:
   IF "M_F_S2-1_1" AND ("CnvF".Sect2_1.I_RFID_2 > 0) THEN "M_F_S2-1_2" := TRUE; END_IF;
END_REGION

REGION Network 46: Mode frw section 2-1 output
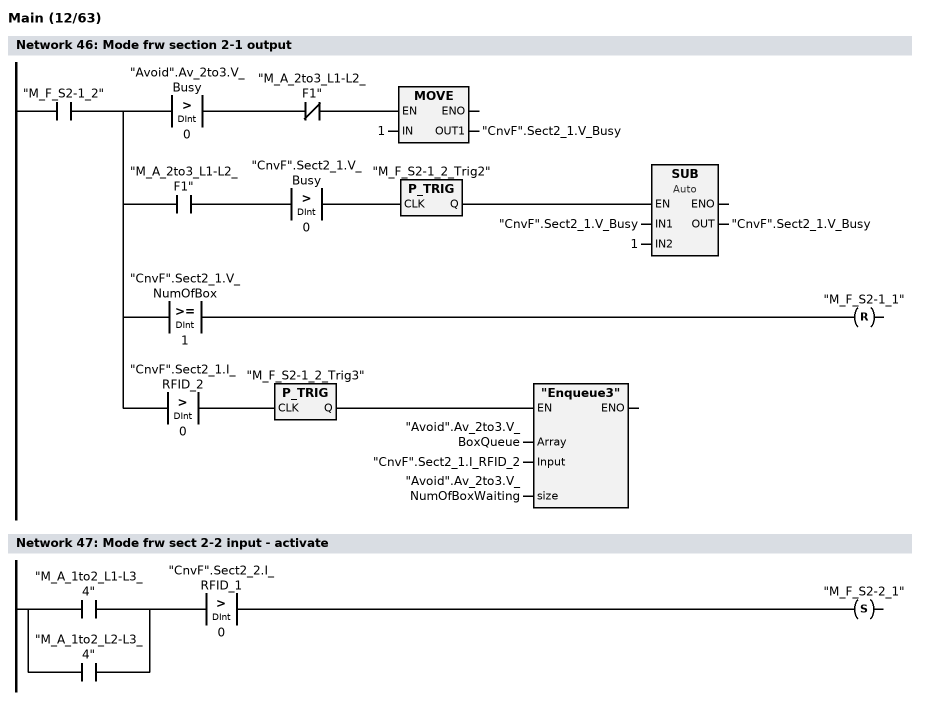
   RUNG wire#powerrail
      Contact( "M_F_S2-1_2" )
      wire#w1
      { S7_Templates := "SrcType := DInt" } GT_Contact(in1 := "Avoid".Av_2to3.V_Busy, in2 := 0)
      I_Contact( "M_A_2to3_L1-L2_F1" )
      Move(in := 1, out1 => "CnvF".Sect2_1.V_Busy)
   END_RUNG
   RUNG wire#w1
      Contact( "M_A_2to3_L1-L2_F1" )
      { S7_Templates := "SrcType := DInt" } GT_Contact(in1 := "CnvF".Sect2_1.V_Busy, in2 := 0)
      P_Trig( "M_F_S2-1_2_Trig2" )
      Sub(in1 := "CnvF".Sect2_1.V_Busy, in2 := 1, out => "CnvF".Sect2_1.V_Busy)
   END_RUNG
   RUNG wire#w1
      { S7_Templates := "SrcType := DInt" } GE_Contact(in1 := "CnvF".Sect2_1.V_NumOfBox, in2 := 1)
      R_Coil( "M_F_S2-1_1" )
   END_RUNG
   RUNG wire#w1
      { S7_Templates := "SrcType := DInt" } GT_Contact(in1 := "CnvF".Sect2_1.I_RFID_2, in2 := 0)
      P_Trig( "M_F_S2-1_2_Trig3" )
      "Enqueue3"("Array" := "Avoid".Av_2to3.V_BoxQueue, Input := "CnvF".Sect2_1.I_RFID_2, size := "Avoid".Av_2to3.V_NumOfBoxWaiting)
   END_RUNG
   // the same network as SCL:
   IF "M_F_S2-1_2" AND ("Avoid".Av_2to3.V_Busy > 0) AND NOT "M_A_2to3_L1-L2_F1" THEN
       "CnvF".Sect2_1.V_Busy := 1;
   END_IF;
   #_w1 := "M_F_S2-1_2" AND "M_A_2to3_L1-L2_F1" AND ("CnvF".Sect2_1.V_Busy > 0);
   #_w2 := #_w1 AND NOT "M_F_S2-1_2_Trig2";   // rising edge
   "M_F_S2-1_2_Trig2" := #_w1;
   IF #_w2 THEN "CnvF".Sect2_1.V_Busy := "CnvF".Sect2_1.V_Busy - 1; END_IF;
   IF "M_F_S2-1_2" AND ("CnvF".Sect2_1.V_NumOfBox >= 1) THEN "M_F_S2-1_1" := FALSE; END_IF;
   #_w3 := "M_F_S2-1_2" AND ("CnvF".Sect2_1.I_RFID_2 > 0);
   #_w4 := #_w3 AND NOT "M_F_S2-1_2_Trig3";   // rising edge
   "M_F_S2-1_2_Trig3" := #_w3;
   IF #_w4 THEN
       "Enqueue3"("Array" := "Avoid".Av_2to3.V_BoxQueue,
                  Input := "CnvF".Sect2_1.I_RFID_2,
                  size := "Avoid".Av_2to3.V_NumOfBoxWaiting);
   END_IF;
END_REGION

REGION Network 47: Mode frw sect 2-2 input - activate
   RUNG wire#powerrail
      Contact( "M_A_1to2_L1-L3_4" )
      wire#w1
      { S7_Templates := "SrcType := DInt" } GT_Contact(in1 := "CnvF".Sect2_2.I_RFID_1, in2 := 0)
      S_Coil( "M_F_S2-2_1" )
   END_RUNG
   RUNG wire#powerrail
      Contact( "M_A_1to2_L2-L3_4" )
   END_RUNG wire#w1
   // the same network as SCL:
   IF ("M_A_1to2_L1-L3_4" OR "M_A_1to2_L2-L3_4") AND ("CnvF".Sect2_2.I_RFID_1 > 0) THEN
       "M_F_S2-2_1" := TRUE;
   END_IF;
END_REGION

REGION Network 48: Mode frw sect 2-2 input
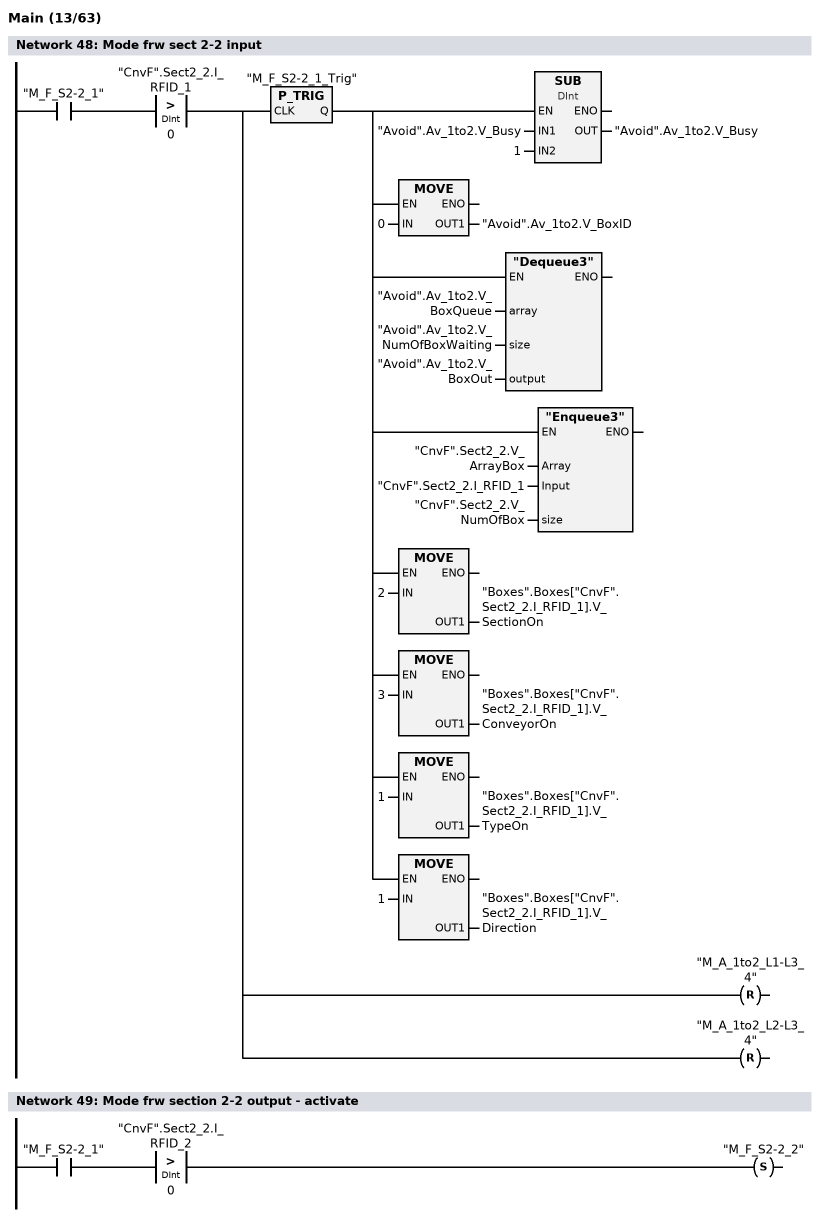
   RUNG wire#powerrail
      Contact( "M_F_S2-2_1" )
      { S7_Templates := "SrcType := DInt" } GT_Contact(in1 := "CnvF".Sect2_2.I_RFID_1, in2 := 0)
      wire#w1
      P_Trig( "M_F_S2-2_1_Trig" )
      wire#w2
      { S7_Templates := "SrcType := DInt" } Sub(in1 := "Avoid".Av_1to2.V_Busy, in2 := 1, out => "Avoid".Av_1to2.V_Busy)
   END_RUNG
   RUNG wire#w2
      Move(in := 0, out1 => "Avoid".Av_1to2.V_BoxID)
   END_RUNG
   RUNG wire#w2
      "Dequeue3"("array" := "Avoid".Av_1to2.V_BoxQueue, size := "Avoid".Av_1to2.V_NumOfBoxWaiting, output := "Avoid".Av_1to2.V_BoxOut)
   END_RUNG
   RUNG wire#w2
      "Enqueue3"("Array" := "CnvF".Sect2_2.V_ArrayBox, Input := "CnvF".Sect2_2.I_RFID_1, size := "CnvF".Sect2_2.V_NumOfBox)
   END_RUNG
   RUNG wire#w2
      Move(in := 2, out1 => "Boxes".Boxes["CnvF".Sect2_2.I_RFID_1].V_SectionOn)
   END_RUNG
   RUNG wire#w2
      Move(in := 3, out1 => "Boxes".Boxes["CnvF".Sect2_2.I_RFID_1].V_ConveyorOn)
   END_RUNG
   RUNG wire#w2
      Move(in := 1, out1 => "Boxes".Boxes["CnvF".Sect2_2.I_RFID_1].V_TypeOn)
   END_RUNG
   RUNG wire#w2
      Move(in := 1, out1 => "Boxes".Boxes["CnvF".Sect2_2.I_RFID_1].V_Direction)
   END_RUNG
   RUNG wire#w1
      R_Coil( "M_A_1to2_L1-L3_4" )
   END_RUNG
   RUNG wire#w1
      R_Coil( "M_A_1to2_L2-L3_4" )
   END_RUNG
   // the same network as SCL:
   #_w1 := "M_F_S2-2_1" AND ("CnvF".Sect2_2.I_RFID_1 > 0);
   #_w2 := #_w1 AND NOT "M_F_S2-2_1_Trig";   // rising edge
   "M_F_S2-2_1_Trig" := #_w1;
   IF #_w2 THEN
       "Avoid".Av_1to2.V_Busy := "Avoid".Av_1to2.V_Busy - 1;
       "Avoid".Av_1to2.V_BoxID := 0;
       "Dequeue3"("array" := "Avoid".Av_1to2.V_BoxQueue,
                  size := "Avoid".Av_1to2.V_NumOfBoxWaiting,
                  output := "Avoid".Av_1to2.V_BoxOut);
       "Enqueue3"("Array" := "CnvF".Sect2_2.V_ArrayBox,
                  Input := "CnvF".Sect2_2.I_RFID_1,
                  size := "CnvF".Sect2_2.V_NumOfBox);
       "Boxes".Boxes["CnvF".Sect2_2.I_RFID_1].V_SectionOn := 2;
       "Boxes".Boxes["CnvF".Sect2_2.I_RFID_1].V_ConveyorOn := 3;
       "Boxes".Boxes["CnvF".Sect2_2.I_RFID_1].V_TypeOn := 1;
       "Boxes".Boxes["CnvF".Sect2_2.I_RFID_1].V_Direction := 1;
   END_IF;
   IF #_w1 THEN
       "M_A_1to2_L1-L3_4" := FALSE;
       "M_A_1to2_L2-L3_4" := FALSE;
   END_IF;
END_REGION

REGION Network 49: Mode frw section 2-2 output - activate
   RUNG wire#powerrail
      Contact( "M_F_S2-2_1" )
      { S7_Templates := "SrcType := DInt" } GT_Contact(in1 := "CnvF".Sect2_2.I_RFID_2, in2 := 0)
      S_Coil( "M_F_S2-2_2" )
   END_RUNG
   // the same network as SCL:
   IF "M_F_S2-2_1" AND ("CnvF".Sect2_2.I_RFID_2 > 0) THEN "M_F_S2-2_2" := TRUE; END_IF;
END_REGION

REGION Network 50: Mode frw section 2-2 output
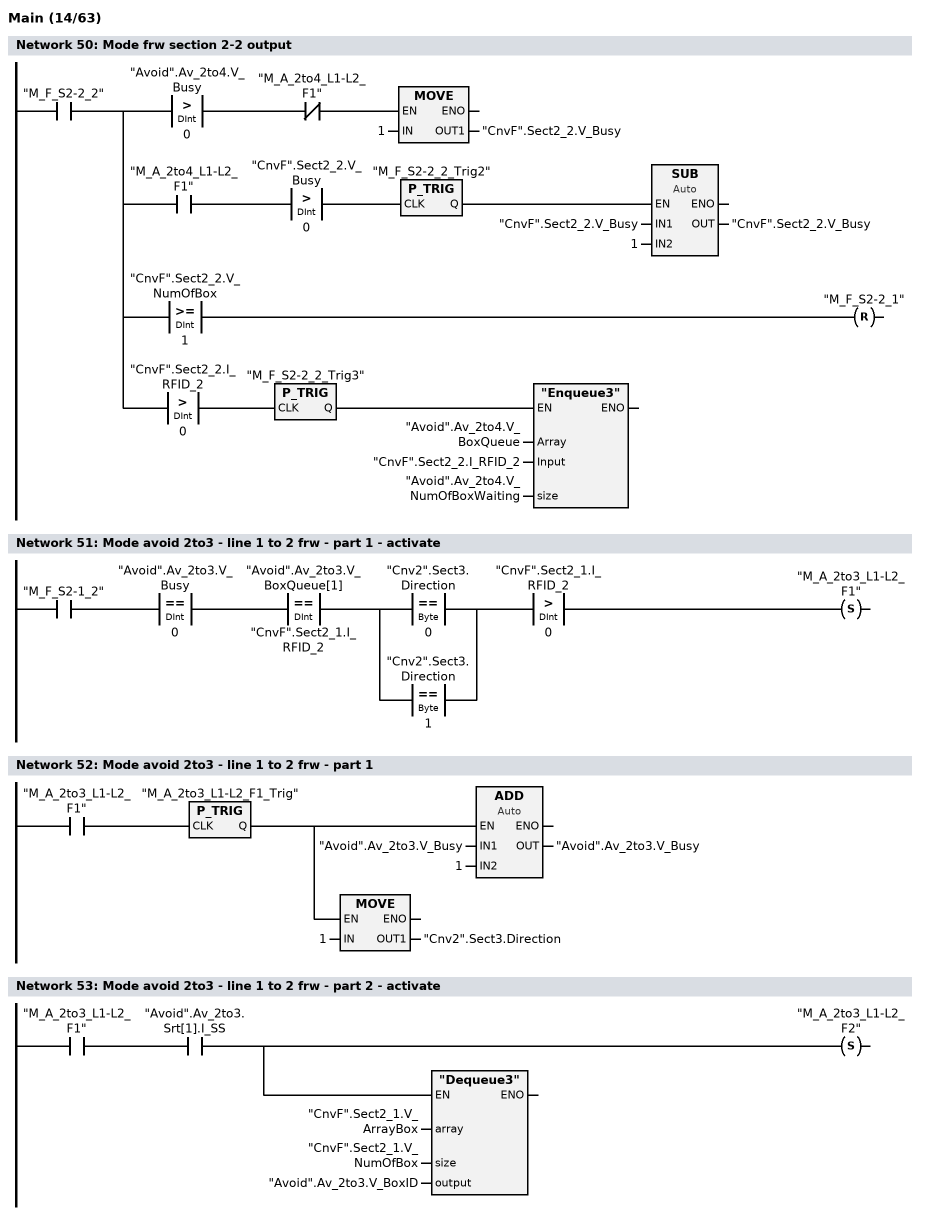
   RUNG wire#powerrail
      Contact( "M_F_S2-2_2" )
      wire#w1
      { S7_Templates := "SrcType := DInt" } GT_Contact(in1 := "Avoid".Av_2to4.V_Busy, in2 := 0)
      I_Contact( "M_A_2to4_L1-L2_F1" )
      Move(in := 1, out1 => "CnvF".Sect2_2.V_Busy)
   END_RUNG
   RUNG wire#w1
      Contact( "M_A_2to4_L1-L2_F1" )
      { S7_Templates := "SrcType := DInt" } GT_Contact(in1 := "CnvF".Sect2_2.V_Busy, in2 := 0)
      P_Trig( "M_F_S2-2_2_Trig2" )
      Sub(in1 := "CnvF".Sect2_2.V_Busy, in2 := 1, out => "CnvF".Sect2_2.V_Busy)
   END_RUNG
   RUNG wire#w1
      { S7_Templates := "SrcType := DInt" } GE_Contact(in1 := "CnvF".Sect2_2.V_NumOfBox, in2 := 1)
      R_Coil( "M_F_S2-2_1" )
   END_RUNG
   RUNG wire#w1
      { S7_Templates := "SrcType := DInt" } GT_Contact(in1 := "CnvF".Sect2_2.I_RFID_2, in2 := 0)
      P_Trig( "M_F_S2-2_2_Trig3" )
      "Enqueue3"("Array" := "Avoid".Av_2to4.V_BoxQueue, Input := "CnvF".Sect2_2.I_RFID_2, size := "Avoid".Av_2to4.V_NumOfBoxWaiting)
   END_RUNG
   // the same network as SCL:
   IF "M_F_S2-2_2" AND ("Avoid".Av_2to4.V_Busy > 0) AND NOT "M_A_2to4_L1-L2_F1" THEN
       "CnvF".Sect2_2.V_Busy := 1;
   END_IF;
   #_w1 := "M_F_S2-2_2" AND "M_A_2to4_L1-L2_F1" AND ("CnvF".Sect2_2.V_Busy > 0);
   #_w2 := #_w1 AND NOT "M_F_S2-2_2_Trig2";   // rising edge
   "M_F_S2-2_2_Trig2" := #_w1;
   IF #_w2 THEN "CnvF".Sect2_2.V_Busy := "CnvF".Sect2_2.V_Busy - 1; END_IF;
   IF "M_F_S2-2_2" AND ("CnvF".Sect2_2.V_NumOfBox >= 1) THEN "M_F_S2-2_1" := FALSE; END_IF;
   #_w3 := "M_F_S2-2_2" AND ("CnvF".Sect2_2.I_RFID_2 > 0);
   #_w4 := #_w3 AND NOT "M_F_S2-2_2_Trig3";   // rising edge
   "M_F_S2-2_2_Trig3" := #_w3;
   IF #_w4 THEN
       "Enqueue3"("Array" := "Avoid".Av_2to4.V_BoxQueue,
                  Input := "CnvF".Sect2_2.I_RFID_2,
                  size := "Avoid".Av_2to4.V_NumOfBoxWaiting);
   END_IF;
END_REGION

REGION Network 51: Mode avoid 2to3 - line 1 to 2 frw - part 1 - activate
   RUNG wire#powerrail
      Contact( "M_F_S2-1_2" )
      { S7_Templates := "SrcType := DInt" } EQ_Contact(in1 := "Avoid".Av_2to3.V_Busy, in2 := 0)
      { S7_Templates := "SrcType := DInt" } EQ_Contact(in1 := "Avoid".Av_2to3.V_BoxQueue[1], in2 := "CnvF".Sect2_1.I_RFID_2)
      wire#w1
      { S7_Templates := "SrcType := Byte" } EQ_Contact(in1 := "Cnv2".Sect3.Direction, in2 := 0)
      wire#w2
      { S7_Templates := "SrcType := DInt" } GT_Contact(in1 := "CnvF".Sect2_1.I_RFID_2, in2 := 0)
      S_Coil( "M_A_2to3_L1-L2_F1" )
   END_RUNG
   RUNG wire#w1
      { S7_Templates := "SrcType := Byte" } EQ_Contact(in1 := "Cnv2".Sect3.Direction, in2 := 1)
   END_RUNG wire#w2
   // the same network as SCL:
   IF "M_F_S2-1_2" AND ("Avoid".Av_2to3.V_Busy = 0) AND ("Avoid".Av_2to3.V_BoxQueue[1] = "CnvF".Sect2_1.I_RFID_2) AND (("Cnv2".Sect3.Direction = 0) OR ("Cnv2".Sect3.Direction = 1)) AND ("CnvF".Sect2_1.I_RFID_2 > 0) THEN
       "M_A_2to3_L1-L2_F1" := TRUE;
   END_IF;
END_REGION

REGION Network 52: Mode avoid 2to3 - line 1 to 2 frw - part 1
   RUNG wire#powerrail
      Contact( "M_A_2to3_L1-L2_F1" )
      P_Trig( "M_A_2to3_L1-L2_F1_Trig" )
      wire#w1
      Add(in1 := "Avoid".Av_2to3.V_Busy, in2 := 1, out => "Avoid".Av_2to3.V_Busy)
   END_RUNG
   RUNG wire#w1
      Move(in := 1, out1 => "Cnv2".Sect3.Direction)
   END_RUNG
   // the same network as SCL:
   #_w1 := "M_A_2to3_L1-L2_F1" AND NOT "M_A_2to3_L1-L2_F1_Trig";   // rising edge
   "M_A_2to3_L1-L2_F1_Trig" := "M_A_2to3_L1-L2_F1";
   IF #_w1 THEN
       "Avoid".Av_2to3.V_Busy := "Avoid".Av_2to3.V_Busy + 1;
       "Cnv2".Sect3.Direction := 1;
   END_IF;
END_REGION

REGION Network 53: Mode avoid 2to3 - line 1 to 2 frw - part 2 - activate
   RUNG wire#powerrail
      Contact( "M_A_2to3_L1-L2_F1" )
      Contact( "Avoid".Av_2to3.Srt[1].I_SS )
      wire#w1
      S_Coil( "M_A_2to3_L1-L2_F2" )
   END_RUNG
   RUNG wire#w1
      "Dequeue3"("array" := "CnvF".Sect2_1.V_ArrayBox, size := "CnvF".Sect2_1.V_NumOfBox, output := "Avoid".Av_2to3.V_BoxID)
   END_RUNG
   // the same network as SCL:
   IF "M_A_2to3_L1-L2_F1" AND "Avoid".Av_2to3.Srt[1].I_SS THEN
       "M_A_2to3_L1-L2_F2" := TRUE;
       "Dequeue3"("array" := "CnvF".Sect2_1.V_ArrayBox,
                  size := "CnvF".Sect2_1.V_NumOfBox,
                  output := "Avoid".Av_2to3.V_BoxID);
   END_IF;
END_REGION

REGION Network 54: Mode avoid 2to3 - line 1 to 2 frw - part 2
